	CASE iTagI OF
		1:
			IF i < DINT_TO_INT(UPPER_BOUND(stEmergencias, 1)) THEN
				RefEmer1 REF= stEmergencias[i].En.xEmergenciaOK;
			ELSE
				RefEmer1 REF= Verdadeiro;
			END_IF
		2:
			IF i < DINT_TO_INT(UPPER_BOUND(stEmergencias, 1)) THEN
				RefEmer2 REF= stEmergencias[i].En.xEmergenciaOK;
			ELSE
				RefEmer2 REF= Verdadeiro;
			END_IF		
		3:
			IF i < DINT_TO_INT(UPPER_BOUND(stEmergencias, 1)) THEN
				RefEmer3 REF= stEmergencias[i].En.xEmergenciaOK;
			ELSE
				RefEmer3 REF= Verdadeiro;
			END_IF
		4:
			IF i < DINT_TO_INT(UPPER_BOUND(stEmergencias, 1)) THEN
				RefEmer4 REF= stEmergencias[i].En.xEmergenciaOK;
			ELSE
				RefEmer4 REF= Verdadeiro;
			END_IF
		
	END_CASE
		
END_FOR

GeraEmergencias := TRUE;
END_METHOD

METHOD PRIVATE GeraNomeInterlock : BOOL
VAR_INPUT
	index : INT;
END_VAR
VAR
	sAux : ARRAY[1..20] OF STRING(255);
	i : INT;
END_VAR


IF stMotor[index].BancoDeDados.IT1A <> '' THEN
	
	IF stMotor[index].BancoDeDados.InvIT1A <> 0 THEN
		IF __ISVALIDREF(RefIT1A) THEN		
			IF (RefIT1A) THEN
				sAux[1] := 'NF(';
			ELSE
				sAux[1] := '*NF*(';
			END_IF
		END_IF
	ELSE
		IF __ISVALIDREF(RefIT1A) THEN	
			IF (RefIT1A) THEN
				sAux[1] := '*NA*(';
			ELSE
				sAux[1] := 'NA(';
			END_IF
		END_IF
	END_IF
	
	IF __ISVALIDREF(RefIT1A) THEN	
		IF (RefIT1A) THEN
			sAux[2] := CONCAT(CONCAT('*',(stMotor[index].BancoDeDados.IT1A)),'*');
		ELSE
			sAux[2] := (stMotor[index].BancoDeDados.IT1A);
		END_IF
	END_IF
	
	sAux[3] := 	')';

	IF stMotor[index].BancoDeDados.IT1B <> '' THEN
		IF stMotor[index].BancoDeDados.OPIT1 <> 0 THEN
			sAux[4] := ' E ';
		ELSE
			sAux[4] := 	' OU ';
		END_IF

		IF stMotor[index].BancoDeDados.InvIT1B <> 0 THEN
			IF __ISVALIDREF(RefIT1B) THEN
				IF (RefIT1B) THEN
					sAux[5] := 'NF(';
				ELSE
					sAux[5] := '*NF*(';
				END_IF
			END_IF
		ELSE
			IF __ISVALIDREF(RefIT1B) THEN
				IF (RefIT1B) THEN
					sAux[5] := '*NA*(';
				ELSE
					sAux[5] := 'NA(';
				END_IF
			END_IF
		END_IF
		
		IF __ISVALIDREF(RefIT1B) THEN
			IF (RefIT1B) THEN
				sAux[6] := CONCAT(CONCAT('*',(stMotor[index].BancoDeDados.IT1B)),'*');
			ELSE
				sAux[6] := (stMotor[index].BancoDeDados.IT1B);
			END_IF
		END_IF
		sAux[7] := 	') ';
	END_IF
ELSE
	stMotor[index].En.sInterLock_1 := '';
END_IF

stMotor[index].En.sInterLock_1 := F_ConcatArray(sAux);

FOR i := 1 TO 20 DO
	sAux[i] := '';
END_FOR


IF stMotor[index].BancoDeDados.IT2A <> '' THEN
	
	IF stMotor[index].BancoDeDados.InvIT2A <> 0 THEN
		IF __ISVALIDREF(RefIT2A) THEN		
			IF (RefIT2A) THEN
				sAux[1] := 'NF(';
			ELSE
				sAux[1] := '*NF*(';
			END_IF
		END_IF
	ELSE
		IF __ISVALIDREF(RefIT2A) THEN	
			IF (RefIT2A) THEN
				sAux[1] := '*NA*(';
			ELSE
				sAux[1] := 'NA(';
			END_IF
		END_IF
	END_IF
	
	IF __ISVALIDREF(RefIT2A) THEN	
		IF (RefIT2A) THEN
			sAux[2] := CONCAT(CONCAT('*',(stMotor[index].BancoDeDados.IT2A)),'*');
		ELSE
			sAux[2] := (stMotor[index].BancoDeDados.IT2A);
		END_IF
	END_IF
	
	sAux[3] := 	')';

	IF stMotor[index].BancoDeDados.IT2B <> '' THEN
		IF stMotor[index].BancoDeDados.OPIT2 <> 0 THEN
			sAux[4] := ' E ';
		ELSE
			sAux[4] := 	' OU ';
		END_IF

		IF stMotor[index].BancoDeDados.InvIT2B <> 0 THEN
			IF __ISVALIDREF(RefIT2B) THEN
				IF (RefIT2B) THEN
					sAux[5] := 'NF(';
				ELSE
					sAux[5] := '*NF*(';
				END_IF
			END_IF
		ELSE
			IF __ISVALIDREF(RefIT2B) THEN
				IF (RefIT2B) THEN
					sAux[5] := '*NA*(';
				ELSE
					sAux[5] := 'NA(';
				END_IF
			END_IF
		END_IF
		
		IF __ISVALIDREF(RefIT2B) THEN
			IF (RefIT2B) THEN
				sAux[6] := CONCAT(CONCAT('*',(stMotor[index].BancoDeDados.IT2B)),'*');
			ELSE
				sAux[6] := (stMotor[index].BancoDeDados.IT2B);
			END_IF
		END_IF
		sAux[7] := 	') ';
	END_IF
ELSE
	stMotor[index].En.sInterLock_2 := '';
END_IF

stMotor[index].En.sInterLock_2 := F_ConcatArray(sAux);

FOR i := 1 TO 20 DO
	sAux[i] := '';
END_FOR


IF stMotor[index].BancoDeDados.IT3A <> '' THEN
	
	IF stMotor[index].BancoDeDados.InvIT3A <> 0 THEN
		IF __ISVALIDREF(RefIT3A) THEN		
			IF (RefIT3A) THEN
				sAux[1] := 'NF(';
			ELSE
				sAux[1] := '*NF*(';
			END_IF
		END_IF
	ELSE
		IF __ISVALIDREF(RefIT3A) THEN	
			IF (RefIT3A) THEN
				sAux[1] := '*NA*(';
			ELSE
				sAux[1] := 'NA(';
			END_IF
		END_IF
	END_IF
	
	IF __ISVALIDREF(RefIT3A) THEN	
		IF (RefIT3A) THEN
			sAux[2] := CONCAT(CONCAT('*',(stMotor[index].BancoDeDados.IT3A)),'*');
		ELSE
			sAux[2] := (stMotor[index].BancoDeDados.IT3A);
		END_IF
	END_IF
	
	sAux[3] := 	')';

	IF stMotor[index].BancoDeDados.IT3B <> '' THEN
		IF stMotor[index].BancoDeDados.OPIT3 <> 0 THEN
			sAux[4] := ' E ';
		ELSE
			sAux[4] := 	' OU ';
		END_IF

		IF stMotor[index].BancoDeDados.InvIT3B <> 0 THEN
			IF __ISVALIDREF(RefIT3B) THEN
				IF (RefIT3B) THEN
					sAux[5] := 'NF(';
				ELSE
					sAux[5] := '*NF*(';
				END_IF
			END_IF
		ELSE
			IF __ISVALIDREF(RefIT3B) THEN
				IF (RefIT3B) THEN
					sAux[5] := '*NA*(';
				ELSE
					sAux[5] := 'NA(';
				END_IF
			END_IF
		END_IF
		
		IF __ISVALIDREF(RefIT3B) THEN
			IF (RefIT3B) THEN
				sAux[6] := CONCAT(CONCAT('*',(stMotor[index].BancoDeDados.IT3B)),'*');
			ELSE
				sAux[6] := (stMotor[index].BancoDeDados.IT3B);
			END_IF
		END_IF
		sAux[7] := 	') ';
	END_IF
ELSE
	stMotor[index].En.sInterLock_3 := '';
END_IF

stMotor[index].En.sInterLock_3 := F_ConcatArray(sAux);

FOR i := 1 TO 20 DO
	sAux[i] := '';
END_FOR


IF stMotor[index].BancoDeDados.IT4A <> '' THEN
	
	IF stMotor[index].BancoDeDados.InvIT4A <> 0 THEN
		IF __ISVALIDREF(RefIT4A) THEN		
			IF (RefIT4A) THEN
				sAux[1] := 'NF(';
			ELSE
				sAux[1] := '*NF*(';
			END_IF
		END_IF
	ELSE
		IF __ISVALIDREF(RefIT4A) THEN	
			IF (RefIT4A) THEN
				sAux[1] := '*NA*(';
			ELSE
				sAux[1] := 'NA(';
			END_IF
		END_IF
	END_IF
	
	IF __ISVALIDREF(RefIT4A) THEN	
		IF (RefIT4A) THEN
			sAux[2] := CONCAT(CONCAT('*',(stMotor[index].BancoDeDados.IT4A)),'*');
		ELSE
			sAux[2] := (stMotor[index].BancoDeDados.IT4A);
		END_IF
	END_IF
	
	sAux[3] := 	')';

	IF stMotor[index].BancoDeDados.IT4B <> '' THEN
		IF stMotor[index].BancoDeDados.OPIT4 <> 0 THEN
			sAux[4] := ' E ';
		ELSE
			sAux[4] := 	' OU ';
		END_IF

		IF stMotor[index].BancoDeDados.InvIT4B <> 0 THEN
			IF __ISVALIDREF(RefIT4B) THEN
				IF (RefIT4B) THEN
					sAux[5] := 'NF(';
				ELSE
					sAux[5] := '*NF*(';
				END_IF
			END_IF
		ELSE
			IF __ISVALIDREF(RefIT4B) THEN
				IF (RefIT4B) THEN
					sAux[5] := '*NA*(';
				ELSE
					sAux[5] := 'NA(';
				END_IF
			END_IF
		END_IF
		
		IF __ISVALIDREF(RefIT4B) THEN
			IF (RefIT4B) THEN
				sAux[6] := CONCAT(CONCAT('*',(stMotor[index].BancoDeDados.IT4B)),'*');
			ELSE
				sAux[6] := (stMotor[index].BancoDeDados.IT4B);
			END_IF
		END_IF
		sAux[7] := 	') ';
	END_IF
ELSE
	stMotor[index].En.sInterLock_4 := '';
END_IF

stMotor[index].En.sInterLock_4 := F_ConcatArray(sAux);

FOR i := 1 TO 20 DO
	sAux[i] := '';
END_FOR







GeraNomeInterlock := true;
END_METHOD

METHOD PRIVATE LinkaOsNaoInterlock : BOOL
VAR_INPUT
END_VAR
//Se inverte
IF EstruturaBanco[0].InvIT1A = 1 THEN
	RefInvIT1A REF= Verdadeiro;
ELSE
	RefInvIT1A REF= FALSO;
END_IF

//Operação feita
IF EstruturaBanco[0].OPIT1 = 1 THEN
	RefOPIT1 REF= Verdadeiro;
ELSE
	RefOPIT1 REF= FALSO;
END_IF

//Se inverte o 1B
IF EstruturaBanco[0].InvIT1B = 1 THEN
	RefInvIT1B REF= Verdadeiro;
ELSE
	RefInvIT1B REF= FALSO;
END_IF

//Se inverte
IF EstruturaBanco[0].InvIT2A = 1 THEN
	RefInvIT2A REF= Verdadeiro;
ELSE
	RefInvIT2A REF= FALSO;
END_IF

//Operação feita
IF EstruturaBanco[0].OPIT2 = 1 THEN
	RefOPIT2 REF= Verdadeiro;
ELSE
	RefOPIT2 REF= FALSO;
END_IF

//Se inverte o 2B
IF EstruturaBanco[0].InvIT2B = 1 THEN
	RefInvIT2B REF= Verdadeiro;
ELSE
	RefInvIT2B REF= FALSO;
END_IF

//Se inverte
IF EstruturaBanco[0].InvIT3A = 1 THEN
	RefInvIT3A REF= Verdadeiro;
ELSE
	RefInvIT3A REF= FALSO;
END_IF

//Operação feita
IF EstruturaBanco[0].OPIT3 = 1 THEN
	RefOPIT3 REF= Verdadeiro;
ELSE
	RefOPIT3 REF= FALSO;
END_IF

//Se inverte o 3B
IF EstruturaBanco[0].InvIT3B = 1 THEN
	RefInvIT3B REF= Verdadeiro;
ELSE
	RefInvIT3B REF= FALSO;
END_IF

//Se inverte
IF EstruturaBanco[0].InvIT4A = 1 THEN
	RefInvIT4A REF= Verdadeiro;
ELSE
	RefInvIT4A REF= FALSO;
END_IF

//Operação feita
IF EstruturaBanco[0].OPIT4 = 1 THEN
	RefOPIT4 REF= Verdadeiro;
ELSE
	RefOPIT4 REF= FALSO;
END_IF

//Se inverte o 4B
IF EstruturaBanco[0].InvIT4B = 1 THEN
	RefInvIT4B REF= Verdadeiro;
ELSE
	RefInvIT4B REF= FALSO;
END_IF
END_METHOD

METHOD PRIVATE MudouNoMotor : BOOL
VAR_INPUT
	Atual		: Teknike_Partidas.ST_ConfigMotorDB;
	Anterior	: Teknike_Partidas.ST_ConfigMotorDB;
END_VAR
VAR
	xMudouNome : BOOL;
	iTamanhoComecaFuncao : INT;
END_VAR

xMudouNome := (CONCAT(CONCAT(stMotor[iIndexMotor].BancoDeDados.Tag, ' - '), stMotor[iIndexMotor].BancoDeDados.Funcao))
				<> stMotor[iIndexMotor].Config.sNome_Funcao;

IF xMudouNome AND NOT (Anterior.Tag <> Atual.Tag OR ((Anterior.Funcao <> Atual.Funcao) AND Atual.Funcao <> '')) THEN
	IF (Anterior.Funcao <> Atual.Funcao) AND (Atual.Funcao = '' OR stMotor[iIndexMotor].Config.sNome_Funcao = '') THEN
		stMotor[iIndexMotor].Config.sNome_Funcao := concat(stMotor[iIndexMotor].BancoDeDados.Tag,stMotor[iIndexMotor].BancoDeDados.Funcao);
	END_IF
	iTamanhoComecaFuncao								:= LEN(stMotor[iIndexMotor].Config.sNome_Funcao) - (LEN(Atual.Tag) + 3);
	stMotor[iIndexMotor].BancoDeDados.Funcao	:= RIGHT(STR := stMotor[iIndexMotor].Config.sNome_Funcao, SIZE := iTamanhoComecaFuncao);
END_IF

MudouNoMotor := 	Anterior.InvIT1A <> Atual.InvIT1A
					OR Anterior.IT1A <> Atual.IT1A
					OR Anterior.OPIT1 <> Atual.OPIT1
					OR Anterior.InvIT1B <> Atual.InvIT1B
					OR Anterior.IT1B <> Atual.IT1B
					OR Anterior.InvIT2A <> Atual.InvIT2A
					OR Anterior.IT2A <> Atual.IT2A
					OR Anterior.OPIT2 <> Atual.OPIT2
					OR Anterior.InvIT2B <> Atual.InvIT2B
					OR Anterior.IT2B <> Atual.IT2B
					OR Anterior.InvIT3A <> Atual.InvIT3A
					OR Anterior.IT3A <> Atual.IT3A
					OR Anterior.OPIT3 <> Atual.OPIT3
					OR Anterior.InvIT3B <> Atual.InvIT3B
					OR Anterior.IT3B <> Atual.IT3B
					OR Anterior.InvIT4A <> Atual.InvIT4A
					OR Anterior.IT4A <> Atual.IT4A
					OR Anterior.OPIT4 <> Atual.OPiT4
					OR Anterior.InvIT4B <> Atual.InvIT4B
					OR Anterior.IT4B <> Atual.IT4B
					OR Anterior.Emerg1 <> Atual.Emerg1
					OR Anterior.Emerg2 <> Atual.Emerg2
					OR Anterior.Emerg3 <> Atual.Emerg3
					OR Anterior.Emerg4 <> Atual.Emerg4
					OR xMudouNome;
END_METHOD

ACTION TrocaEstadoLeitura:

//EstadoAtual := ExecutaInterlocks;

CASE EstadoAtual OF

	enum_MaquinaConfigPartidaDB.Esperando:
		xOcupado := FALSE;
		rtAtualiza(CLK := xLe, Q =>);

		//controla pra nao ficar muitos acessando o banco 
		//IF rtAtualiza.q THEN
			IF iMaxAtualizando > iAtualizandoAtual AND xLe THEN
				EstadoAtual	:= enum_MaquinaConfigPartidaDB.LendoEleMesmo;
				xOcupado	:= TRUE;
			//ELSE
			//	xLe := FALSE;
			END_IF	
		//END_IF

		EstruturaAnterior := stMotor[iIndexMotor].BancoDeDados;

	enum_MaquinaConfigPartidaDB.AbreConexao:
		//xOcupado := TRUE;
		
		xTemQueAtualizarSQL := FALSE;//joga pra falso pq so aqui é que realmente ele ta atualizando o SQL
		
		IF fbSqlDatabase.Connect(INT_TO_UDINT(iNumeroDataBase)) THEN
			IF fbSqlDatabase.bError THEN
				{error <'Não conseguiu conectar para ler o banco no bloco FB_ConfigPartidaNoBanco 1'>}
				IF fbSqlDatabase.ipTcResult.nEventId = 1828 THEN
					// se der isso ele nao fica tentando e gerando uma caralhada de erro pq nao tem a lisença
					EstadoAtual := enum_MaquinaConfigPartidaDB.falha;
				ELSE
					EstadoAtual := enum_MaquinaConfigPartidaDB.AbreConexao;
				END_IF
			ELSE
				IF fbSqlDatabase.bConnected THEN
					EstadoAtual := enum_MaquinaConfigPartidaDB.CriaComando;
				END_IF
			END_IF
		END_IF

	enum_MaquinaConfigPartidaDB.CriaComando:
		//xOcupado := TRUE;

		IF fbSqlDatabase.CreateCmd(ADR(fbSqlCommand)) THEN
			IF fbSqlDatabase.bError THEN
				{error <'Não conseguiu criar o comando para ler o banco no bloco FB_ConfigPartidaNoBanco 2'>}
				EstadoAtual := enum_MaquinaConfigPartidaDB.CriaComando;
			ELSE
				EstadoAtual := enum_MaquinaConfigPartidaDB.Gravando;
			END_IF
		END_IF

	enum_MaquinaConfigPartidaDB.Gravando:
		//xOcupado := TRUE;

		IF sCmdUpdate <> '' THEN
			IF fbSQLCommand.Execute(pSQLCmd := ADR(sCmdUpdate), cbSQLCmd := SIZEOF(sCmdUpdate)) THEN
				EstadoAtual	:= enum_MaquinaConfigPartidaDB.FechaConexao;
				sCmdUpdate	:= '';
			END_IF
		END_IF

	enum_MaquinaConfigPartidaDB.FechaConexao:
		//xOcupado := TRUE;

		IF fbSqlDatabase.Disconnect() THEN
			IF fbSqlDatabase.bError THEN
				{error <'Não conseguiu desconectar depois de ler o banco no bloco FB_ConfigPartidaNoBanco 3'>}
				EstadoAtual := enum_MaquinaConfigPartidaDB.FechaConexao;
			ELSE
				xLe			:= TRUE;
				EstadoAtual	:= enum_MaquinaConfigPartidaDB.LendoEleMesmo;
			END_IF
		END_IF

	enum_MaquinaConfigPartidaDB.LendoEleMesmo:
		//xOcupado := TRUE;

		IF NOT xLe THEN
			EstadoAtual := enum_MaquinaConfigPartidaDB.LinkaOsNaoInterlock;
		END_IF

	enum_MaquinaConfigPartidaDB.LinkaOsNaoInterlock:
		//xOcupado			:= TRUE;

		IF __ISVALIDREF(RefInvIT4A) AND __ISVALIDREF(RefOPIT4) AND __ISVALIDREF(RefInvIT4B) THEN
			EstadoAtual	:= enum_MaquinaConfigPartidaDB.ProcuraTag1;
			iTag		:= 1;
		END_IF

	enum_MaquinaConfigPartidaDB.ProcuraTag1:
		//xOcupado			:= TRUE;

		IF __ISVALIDREF(RefIT1A) AND __ISVALIDREF(RefIT2A) AND __ISVALIDREF(RefIT3A) AND __ISVALIDREF(RefIT4A) THEN
			EstadoAtual	:= enum_MaquinaConfigPartidaDB.ProcuraTag2;
			iTag		:= 1;
		END_IF

	enum_MaquinaConfigPartidaDB.ProcuraTag2:
		//xOcupado			:= TRUE;

		IF __ISVALIDREF(RefIT1B) AND __ISVALIDREF(RefIT2B) AND __ISVALIDREF(RefIT3B) AND __ISVALIDREF(RefIT4B) THEN
			EstadoAtual := enum_MaquinaConfigPartidaDB.Gera_sInterlock;
		END_IF

	enum_MaquinaConfigPartidaDB.Gera_sInterlock:
		//xOcupado			:= TRUE;
		EstruturaAnterior	:= stMotor[iIndexMotor].BancoDeDados;
		
		stMotor[iIndexMotor].Config.sNome_Funcao := (CONCAT(CONCAT(stMotor[iIndexMotor].BancoDeDados.Tag,' - '),stMotor[iIndexMotor].BancoDeDados.Funcao));

		IF GeraNomeInterlock(iIndexMotor) THEN
			EstadoAtual := enum_MaquinaConfigPartidaDB.Gera_Emergencia;
		END_IF
		
	enum_MaquinaConfigPartidaDB.Gera_Emergencia:
		IF GeraEmergencias(iIndexMotor) THEN
			EstadoAtual := enum_MaquinaConfigPartidaDB.ExecutaInterlocks;
		END_IF

	enum_MaquinaConfigPartidaDB.ExecutaInterlocks:
		xOcupado := FALSE;
		
		GeraNomeInterlock(iIndexMotor);
		
		rtAtualiza(CLK := xLe, Q =>);

		//controla pra nao ficar muitos acessando o banco 
		IF iMaxAtualizando > iAtualizandoAtual AND xLe THEN
			EstadoAtual	:= enum_MaquinaConfigPartidaDB.LendoEleMesmo;
			xOcupado	:= TRUE;	
		END_IF

		IF xAtualizadoExternamente THEN
			xAtualizadoExternamente	:= FALSE;
			GeraNomeInterlock(iIndexMotor);
			stMotor[iIndexMotor].Config.sNome_Funcao := (CONCAT(CONCAT(stMotor[iIndexMotor].BancoDeDados.Tag,' - '),stMotor[iIndexMotor].BancoDeDados.Funcao));
			EstruturaAnterior		:= stMotor[iIndexMotor].BancoDeDados;
		END_IF
		
		IF MudouNoMotor(stMotor[iIndexMotor].BancoDeDados, EstruturaAnterior) THEN
			xTemQueAtualizarSQL := TRUE;
		END_IF

		IF xTemQueAtualizarSQL AND iMaxAtualizando > iAtualizandoAtual THEN
			EstadoAtual	:= enum_MaquinaConfigPartidaDB.AbreConexao;
			xOcupado	:= TRUE;
		END_IF

		//EstruturaAnterior := stMotor[iIndexMotor].BancoDeDados;

END_CASE
END_ACTION

METHOD PRIVATE ZeraReferencias : BOOL
VAR_INPUT
END_VAR


RefInvIT1A	REF= 0;
IF stMotor[iIndexMotor].BancoDeDados.IT1A <> EstruturaAnterior.IT1A THEN
	RefIT1A	REF= 0;
END_IF
RefOPIT1	REF= 0;
RefInvIT1B	REF= 0;
IF stMotor[iIndexMotor].BancoDeDados.IT1B <> EstruturaAnterior.IT1B THEN
	RefIT1B	REF= 0;
END_IF

RefInvIT2A	REF= 0;
IF stMotor[iIndexMotor].BancoDeDados.IT2A <> EstruturaAnterior.IT2A THEN
	RefIT2A	REF= 0;
END_IF
RefOPIT2	REF= 0;
RefInvIT2B	REF= 0;
IF stMotor[iIndexMotor].BancoDeDados.IT2B <> EstruturaAnterior.IT2B THEN
	RefIT2B	REF= 0;
END_IF

RefInvIT3A	REF= 0;
IF stMotor[iIndexMotor].BancoDeDados.IT3A <> EstruturaAnterior.IT3A THEN
	RefIT3A	REF= 0;
END_IF
RefOPIT3	REF= 0;
RefInvIT3B	REF= 0;
IF stMotor[iIndexMotor].BancoDeDados.IT3B <> EstruturaAnterior.IT3B THEN
	RefIT3B	REF= 0;
END_IF

RefInvIT4A	REF= 0;
IF stMotor[iIndexMotor].BancoDeDados.IT4A <> EstruturaAnterior.IT4A THEN
	RefIT4A	REF= 0;
END_IF
RefOPIT4	REF= 0;
RefInvIT4B	REF= 0;
IF stMotor[iIndexMotor].BancoDeDados.IT4B <> EstruturaAnterior.IT4B THEN
	RefIT4B	REF= 0;
END_IF


RefEmer1	REF= 0;
RefEmer2	REF= 0;
RefEmer3	REF= 0;
RefEmer4	REF= 0;
END_METHOD

END_FUNCTION_BLOCK

// FBs/Intralogistica/Top10SKU/FB_HistogramaSKUsMaisLidas
//{attribute 'hide_all_locals'}
FUNCTION_BLOCK FB_HistogramaSKUsMaisLidas
VAR_INPUT
	sSKU			: STRING;
	xEscreve 		: BOOL;
	xCriaEvento		: BOOL := TRUE;
	xVeOsTop10		: BOOL;
	TempoGuardandoSKUemMinutos : UDINT := 60;
	xCriaTabela		: BOOL;
	iNumeroDataBase	: INT := 1;
	sNomeTabela		: STRING	:= 'TopSKU';
END_VAR
VAR_OUTPUT
	TopSKUs 			: ARRAY[1..10] OF DUT_Top10SKU;
	EstadoEscreve 		: Enum_HistorogramaSKUs := Enum_HistorogramaSKUs.Esperando;
	EstadoEvento 		: Enum_HistorogramaSKUs := Enum_HistorogramaSKUs.Esperando;
	EstadoTOP 			: Enum_HistorogramaSKUs := Enum_HistorogramaSKUs.Esperando;
END_VAR
VAR
	UltimotempoGuardado : UDINT;
	rtCria			: R_TRIG;
	xCria			: BOOL;
	fbPLCDBCreate	: FB_PLCDBCreateEvt(sNetID := '', tTimeout := T#30S);

	ColumnInfo : ARRAY[0..2] OF ST_ColumnInfo := [(sName := 'ID', eType := E_ColumnType.BigInt, nLength := 8, sProperty := 'IDENTITY(1,1)'),
												(sName := 'SKU', eType := E_ColumnType.Integer, nLength := 4),
												(
				sName := 'Timestamp',
					eType := E_ColumnType.DateTime,
					nLength := 4,
					sProperty := 'DEFAULT CURRENT_TIMESTAMP ON UPDATE CURRENT_TIMESTAMP')];



	ColumnNamesLe : ARRAY[0..2] OF STRING(50) := ['ID',
												'SKU',
												'Timestamp'];
	iTamanhoHistorico : DINT;

	i : INT;
	
	fbSqlCommandEscreve		: FB_SQLCommandEvt(sNetID := '', tTimeout := T#30S);
	fbSQLDatabaseEscreve	: FB_SQLDatabaseEvt(sNetID := '', tTimeout := T#30S);
	sCmdEscreve				: STRING(1000);
	xAbertoEscreve 			: BOOL;
	rtEscreve 				: R_TRIG;
	sAuxEscreve				: ARRAY[0..10] OF STRING(255);
	
	fbSqlCommandEvento		: FB_SQLCommandEvt(sNetID := '', tTimeout := T#30S);
	fbSQLDatabaseEvento		: FB_SQLDatabaseEvt(sNetID := '', tTimeout := T#30S);
	sCmdEvento				: STRING(1000);
	xAbertoEvento 			: BOOL;
	rtEvento 				: R_TRIG;
	sAuxEvento				: ARRAY[0..10] OF STRING(255);
	
	
	fbSqlCommandtop			: FB_PLCDBCmdEvt(sNetID := '', tTimeout := T#30S);
	fbSQLDatabaseTOP		: FB_SQLDatabaseEvt(sNetID := '', tTimeout := T#30S);
	sCmdTOP					: STRING(1000);
	xAbertoTOP 				: BOOL;
	rtTOP 					: R_TRIG;
	sAuxTop					: ARRAY[0..10] OF STRING(255);
	stParaTop				: ST_ExpParameter;
	sPara					: STRING(80);
	nRecords				: UDINT;
	LeituraAux				: ARRAY[1..10] OF DUT_Top10SKU;
	
	sMensagemErro1 		: STRING;
	rtComecaEscrever : R_TRIG;
	

END_VAR


IF xLicensaValida651641iih THEN
	
	rtEscreve(CLK:= xEscreve, Q=> );
	rtEvento(CLK:= xCriaEvento OR TempoGuardandoSKUemMinutos <> UltimotempoGuardado, Q=> );
	rtTop(CLK:= xVeOsTop10, Q=> );
	
	UltimotempoGuardado := TempoGuardandoSKUemMinutos;
	
	GeraTabela();
	
	Tabela();
	
	Evento();
	
	Top10();

END_IF

ACTION Evento:

CASE EstadoEvento OF
	 Enum_HistorogramaSKUs.Esperando: //Esperando
		IF rtEvento.q THEN
			IF xAbertoEvento THEN
				EstadoEvento := Enum_HistorogramaSKUs.CriaComando;
			ELSE
				EstadoEvento := Enum_HistorogramaSKUs.AbreConexao;
			END_IF
		END_IF

	Enum_HistorogramaSKUs.AbreConexao: //abre conexao
		IF fbSQLDatabaseEvento.Connect(int_to_udint(iNumeroDataBase)) THEN
			IF fbSQLDatabaseEvento.bError THEN
				IF fbSQLDatabaseEvento.ipTcResult.nEventId = 1828 THEN
					// se der isso ele nao fica tentando e gerando uma caralhada de erro pq nao tem a lisensa
					EstadoEvento := Enum_HistorogramaSKUs.erro;
				ELSE
					EstadoEvento := Enum_HistorogramaSKUs.AbreConexao;
				END_IF
			ELSE
				IF fbSQLDatabaseEvento.bConnected THEN
					EstadoEvento := Enum_HistorogramaSKUs.CriaComando;
					xAbertoEvento := TRUE;
				ELSE
					EstadoEvento := Enum_HistorogramaSKUs.FechaConexao;
					xAbertoEvento := FALSE;
				END_IF
			END_IF
		END_IF
	
	Enum_HistorogramaSKUs.CriaComando:
		IF fbSQLDatabaseEvento.CreateCmd(ADR(fbSqlCommandEvento)) THEN
			IF fbSQLDatabaseEvento.bError THEN
				EstadoEvento := Enum_HistorogramaSKUs.CriaComando;
			ELSE
				EstadoEvento := Enum_HistorogramaSKUs.DeletaEvento;
			END_IF
		END_IF
	
		
	Enum_HistorogramaSKUs.DeletaEvento:
	
		F_LimpaArrayString(sAuxEvento);
	
		sAuxEvento[0] := 'drop event Exclui';
		sAuxEvento[1] := sNomeTabela;
		sAuxEvento[2] := ';';

		sCmdEvento := F_ConcatArray(sAuxEvento);	


		// call functionblock	
		IF fbSqlCommandEvento.Execute(pSQLCmd := ADR(sCmdEvento), cbSQLCmd := SIZEOF(sCmdEvento))THEN
			IF fbSqlCommandEvento.bError THEN
				IF fbSqlCommandEvento.ipTcResult.nEventId = 61 THEN
				// se der isso ele nao fica tentando e gerando uma caralhada de erro pq nao tem a tabela
					EstadoEvento := Enum_HistorogramaSKUs.Esperando;
					xCriaTabela := TRUE;
				ELSE
					EstadoEvento := Enum_HistorogramaSKUs.DeletaEvento;
				END_IF
				sMensagemErro1 := 'Nao conseguiu a tag';
			ELSE
				sMensagemErro1	:= 'Conseguiu a tag';
			END_IF
			EstadoEvento := Enum_HistorogramaSKUs.CriaEvento;
		END_IF
		
	Enum_HistorogramaSKUs.CriaEvento:
	
		F_LimpaArrayString(sAuxEvento);
	
		sAuxEvento[0] := 'CREATE EVENT IF NOT EXISTS Exclui';
		sAuxEvento[1] := sNomeTabela;
		sAuxEvento[2] := ' ON SCHEDULE every 1 minute DO delete from topsku where Timestamp < (NOW() - interval ';
		sAuxEvento[3] := UDINT_TO_STRING(TempoGuardandoSKUemMinutos);
		sAuxEvento[4] := ' minute);';

		 

		sCmdEvento := F_ConcatArray(sAuxEvento);	


		// call functionblock	
		IF fbSqlCommandEvento.Execute(pSQLCmd := ADR(sCmdEvento), cbSQLCmd := SIZEOF(sCmdEvento))THEN
			IF fbSqlCommandEvento.bError THEN
				IF fbSqlCommandEvento.ipTcResult.nEventId = 61 THEN
				// se der isso ele nao fica tentando e gerando uma caralhada de erro pq nao tem a tabela
					EstadoEvento := Enum_HistorogramaSKUs.Esperando;
					xCriaTabela := TRUE;
				ELSE
					EstadoEvento := Enum_HistorogramaSKUs.CriaEvento;
				END_IF
				sMensagemErro1 := 'Nao conseguiu a tag';
			ELSE
				sMensagemErro1	:= 'Conseguiu a tag';
			END_IF
			EstadoEvento := Enum_HistorogramaSKUs.FechaConexao;
			xCriaEvento := FALSE;
		END_IF
		

	Enum_HistorogramaSKUs.FechaConexao: // FechaConexao conexao
		IF fbSQLDatabaseEvento.Disconnect() THEN
			IF NOT fbSQLDatabaseEvento.bError THEN
				EstadoEvento := Enum_HistorogramaSKUs.Esperando;
				xAbertoEvento := FALSE;
			END_IF
		END_IF
END_CASE
END_ACTION

ACTION GeraTabela:

rtCria(CLK := xCriaTabela, Q =>);

IF rtCria.q THEN
	xCria := TRUE;
END_IF

IF xCria THEN
	IF fbPLCDBCreate.Table(
			hDBID := INT_TO_UDINT(iNumeroDataBase),
			sTableName := sNomeTabela,
			pTableCfg := ADR(ColumnInfo),
			cbTableCfg := SIZEOF(ColumnInfo))
	THEN
		xCria := FALSE;
		xCriaTabela := FALSE;
	END_IF

END_IF
END_ACTION

ACTION Tabela:

CASE EstadoEscreve OF
	Enum_HistorogramaSKUs.Esperando: //Esperando
		IF rtEscreve.q THEN
			IF xAbertoEscreve THEN
				EstadoEscreve := Enum_HistorogramaSKUs.CriaComando;
			ELSE
				EstadoEscreve := Enum_HistorogramaSKUs.AbreConexao;
			END_IF
		END_IF

	Enum_HistorogramaSKUs.AbreConexao: //abre conexao
		IF fbSQLDatabaseEscreve.Connect(int_to_udint(iNumeroDataBase)) THEN
			IF fbSQLDatabaseEscreve.bError THEN
				IF fbSQLDatabaseEscreve.ipTcResult.nEventId = 1828 THEN
					// se der isso ele nao fica tentando e gerando uma caralhada de erro pq nao tem a lisensa
					EstadoEscreve := Enum_HistorogramaSKUs.erro;
				ELSE
					EstadoEscreve := Enum_HistorogramaSKUs.AbreConexao;
				END_IF
			ELSE
				IF fbSQLDatabaseEscreve.bConnected THEN
					EstadoEscreve := Enum_HistorogramaSKUs.CriaComando;
					xAbertoEscreve := TRUE;
				ELSE
					EstadoEscreve := Enum_HistorogramaSKUs.FechaConexao;
					xAbertoEscreve := FALSE;
				END_IF
			END_IF
		END_IF
	
	Enum_HistorogramaSKUs.CriaComando:
		IF fbSQLDatabaseEscreve.CreateCmd(ADR(fbSqlCommandEscreve)) THEN
			IF fbSQLDatabaseEscreve.bError THEN
				EstadoEscreve := Enum_HistorogramaSKUs.CriaComando;
			ELSE
				EstadoEscreve := Enum_HistorogramaSKUs.Grava;
			END_IF
		END_IF
	

	Enum_HistorogramaSKUs.Grava: // le o role
	
		F_LimpaArrayString(sAuxEscreve);
	
		sAuxEscreve[0] := 'INSERT INTO ';
		sAuxEscreve[1] := sNomeTabela;
		sAuxEscreve[2] := '(sku) Value ($'';
		sAuxEscreve[3] := sSKU;
		sAuxEscreve[4] := '$');';

		sCmdEscreve := F_ConcatArray(sAuxEscreve);	



		IF fbSqlCommandEscreve.Execute(pSQLCmd := ADR(sCmdEscreve), cbSQLCmd := SIZEOF(sCmdEscreve)) THEN
			IF fbSqlCommandEscreve.bError THEN
				IF fbSqlCommandEscreve.ipTcResult.nEventId = 61 THEN
				// se der isso ele nao fica tentando e gerando uma caralhada de erro pq nao tem a tabela
					EstadoEscreve := Enum_HistorogramaSKUs.Esperando;
					xCriaTabela := TRUE;
				ELSE
					EstadoEscreve := Enum_HistorogramaSKUs.AbreConexao;
				END_IF
				sMensagemErro1 := 'Nao conseguiu a tag';
			ELSE
				sMensagemErro1	:= 'Conseguiu a tag';
			END_IF
			EstadoEscreve := Enum_HistorogramaSKUs.FechaConexao;
			xEscreve := FALSE;
		END_IF
		
	
		

	Enum_HistorogramaSKUs.FechaConexao: // FechaConexao conexao
		IF fbSQLDatabaseEscreve.Disconnect() THEN
			IF NOT fbSQLDatabaseEscreve.bError THEN
				EstadoEscreve := Enum_HistorogramaSKUs.Esperando;
				xAbertoEscreve := FALSE;
			END_IF
		END_IF
END_CASE
END_ACTION

ACTION Top10:

CASE Estadotop OF
	Enum_HistorogramaSKUs.Esperando: //Esperando
		IF rtTop.q THEN
			IF xAbertoTop THEN
				Estadotop := Enum_HistorogramaSKUs.CriaComando;
			ELSE
				Estadotop := Enum_HistorogramaSKUs.AbreConexao;
			END_IF
		END_IF

	Enum_HistorogramaSKUs.AbreConexao: //abre conexao
		IF fbSQLDatabasetop.Connect(int_to_udint(iNumeroDataBase)) THEN
			IF fbSQLDatabasetop.bError THEN
				IF fbSQLDatabasetop.ipTcResult.nEventId = 1828 THEN
					// se der isso ele nao fica tentando e gerando uma caralhada de erro pq nao tem a lisensa
					Estadotop := Enum_HistorogramaSKUs.erro;
				ELSE
					Estadotop := Enum_HistorogramaSKUs.AbreConexao;
				END_IF
			ELSE
				IF fbSQLDatabasetop.bConnected THEN
					Estadotop := Enum_HistorogramaSKUs.Vetop10;
					xAbertotop := TRUE;
				ELSE
					Estadotop := Enum_HistorogramaSKUs.FechaConexao;
					xAbertotop := FALSE;
				END_IF
			END_IF
		END_IF
	
		
	Enum_HistorogramaSKUs.Vetop10:
	
		F_LimpaArrayString(sAuxtop);
	
		sAuxtop[0] := 'SELECT SKU, count(*) FROM ';
		sAuxtop[1] := sNomeTabela;
		sAuxtop[2] := ' GROUP BY SKU ORDER BY count(*) DESC LIMIT 10;';
		 
		sCmdtop := F_ConcatArray(sAuxtop);	
		
		
		stParaTop.eParaType	:= E_ExpParameterType.STRING_;
		stParaTop.nParaSize	:= SIZEOF(sPara);
		stParaTop.sParaName	:= 'Inutil';


		// call functionblock	
		IF fbSqlCommandtop.ExecuteDataReturn(
										hDBID := INT_TO_UDINT(iNumeroDataBase),
										pExpression := ADR(sCmdtop),
										cbExpression := SIZEOF(sCmdtop),
										pData := ADR(sPara),
										cbData := SIZEOF(sPara),
										pParameter := ADR(stParaTop),
										cbParameter := SIZEOF(stParaTop),
										nStartIndex := 0,
										nRecordCount := 10,
										pReturnData := ADR(TopSKUs),
										cbReturnData := SIZEOF(TopSKUs),
										pRecords := ADR(nRecords))
													THEN
			IF fbSqlCommandtop.bError THEN
				IF fbSqlCommandtop.ipTcResult.nEventId = 61 THEN
				// se der isso ele nao fica tentando e gerando uma caralhada de erro pq nao tem a tabela
					Estadotop := Enum_HistorogramaSKUs.Esperando;
					xCriaTabela := TRUE;
				ELSE
					Estadotop := Enum_HistorogramaSKUs.FechaConexao;
				END_IF
				sMensagemErro1 := 'Nao conseguiu a tag';
			ELSE
				sMensagemErro1	:= 'Conseguiu a tag';
			END_IF
			Estadotop := Enum_HistorogramaSKUs.FechaConexao;
			xVeOsTop10 := FALSE;
		END_IF
		

	Enum_HistorogramaSKUs.FechaConexao: // FechaConexao conexao
		IF fbSQLDatabasetop.Disconnect() THEN
			IF NOT fbSQLDatabasetop.bError THEN
				Estadotop := Enum_HistorogramaSKUs.Esperando;
				xAbertotop := FALSE;
			END_IF
		END_IF
END_CASE
END_ACTION

END_FUNCTION_BLOCK

// FBs/MedicaoEnergia/FB_CentroDeCustos2
FUNCTION_BLOCK FB_CentroDeCustos2
VAR_IN_OUT
	Minutos				: ARRAY[*] OF stMinuto;
	Media15Min			: ARRAY[*] OF stMedia15min;
	MediaDia			: ARRAY[*] OF stMediaDia;
	MediaMes			: ARRAY[*] OF stMediaMes;
	PosicaoAtualdos15	: ARRAY[*,*] OF INT;
END_VAR
VAR_INPUT
	xCriaTabelas			: BOOL;				// tenta criar a tabela
	iNumeroDataBase			: INT	:= 1;		// id do database
	iMedidor				: INT;
	sMedidor				: STRING(1000);
	Timestamp				: DT;
	xAtualiza				: BOOL;
	x15minSelecionado		: BOOL;
	xDiaSelecionado			: BOOL;
	xMesSelecionado			: BOOL;
	xAnoSelecionado			: BOOL;
END_VAR
VAR_OUTPUT
	xOcupado 				: BOOL;
	xTodasTabelasCriadas	: BOOL;
	xTerminouLeitura		: BOOL := FALSE;
	sMedidoresSelecionados	: STRING(1000);
END_VAR
VAR
	//Le Valores Centros de Custo
	xAtualizaInterno			: BOOL;
	sCmdEscreve1				: STRING(2000);
	sCmdEscreve2				: STRING(2000);
	sCmdEscreve3				: STRING(2000);
	sCmdEscreve4				: STRING(2000);
	sMensagemErro				: STRING;
	nRecords					: UDINT;
	TagAProcurar				: REAL;
	arString					: ARRAY[0..12] OF STRING(1000);
	diCima						: DINT;
	diBaixo						: DINT;
	i							: INT;
	j							: INT;
	posicao						: INT := 1;
	iEstadoLeitura				: INT := 1;
	minute						: TIMESTRUCT;
	times						: TIMESTRUCT;
	TagAProcurar2				: REAL;
	fbSQLDatabase2				: FB_SQLDatabaseEvt(sNetID := '', tTimeout := T#30S);
	fbPLCDBCmd1					: FB_PLCDBCmdEvt(sNetID := '', tTimeout := T#30S);
	fbPLCDBCmd2					: FB_PLCDBCmdEvt(sNetID := '', tTimeout := T#30S);
	fbPLCDBCmd3					: FB_PLCDBCmdEvt(sNetID := '', tTimeout := T#30S);
	fbPLCDBCmd4					: FB_PLCDBCmdEvt(sNetID := '', tTimeout := T#30S);
	stPara2						: ST_ExpParameter;
	MinutosAtuais				: ARRAY[1..15] OF INT;
	EstruturaBancoMinuto		: ARRAY[1..900] OF stMinuto;
	EstruturaBancoMedia15min	: ARRAY[1..5760] OF stMedia15min;
	EstruturaBancoMediaDia		: ARRAY[1..1860] OF stMediaDia;
	EstruturaBancoMediaMes		: ARRAY[1..720] OF stMediaMes;
	OrganizaEstrutura			: ARRAY[0..132] OF stOrganizaDados;
	rtLeitura1					: R_TRIG;
	rtLeitura2					: R_TRIG;
	rtLeitura3					: R_TRIG;
	rtLeitura4					: R_TRIG;
	rtLeitura5					: R_TRIG;
END_VAR

rtLeitura1(CLK:= xAtualiza, Q=> );
rtLeitura2(CLK:= x15minSelecionado, Q=> );
rtLeitura3(CLK:= xDiaSelecionado, Q=> );
rtLeitura4(CLK:= xMesSelecionado, Q=> );
rtLeitura5(CLK:= xAnoSelecionado, Q=> );

IF rtLeitura1.Q OR rtLeitura2.Q OR rtLeitura3.Q OR rtLeitura4.Q OR rtLeitura5.Q THEN
	xAtualizaInterno 	:= TRUE;
	xTerminouLeitura	:= FALSE;
END_IF

sMedidoresSelecionados := sMedidor;

LeValores();

ACTION LeValores:
CASE iEstadoLeitura OF
	1: //Esperando
		IF xAtualizaInterno THEN
			iEstadoLeitura := 2;
		END_IF

	2: //abre conexao
		IF fbSQLDatabase2.Connect(INT_TO_UDINT(iNumeroDataBase)) THEN
			IF fbSQLDatabase2.bError THEN
				IF fbSQLDatabase2.ipTcResult.ipSourceInfo.sName = 'ADSERR_DEVICE_LICENSENOTFOUND' THEN
					// se der isso ele nao fica tentando e gerando uma caralhada de erro pq nao tem a lisença
					iEstadoLeitura := 0;
				ELSE
					iEstadoLeitura := 2;
				END_IF
			ELSE
				IF fbSQLDatabase2.bConnected THEN
					iEstadoLeitura := 3;
				END_IF
			END_IF
		END_IF

	3: 
		IF x15minSelecionado THEN
			// Le os Minutos
			stPara2.eParaType	:= E_ExpParameterType.Float32;
			stPara2.nParaSize	:= SIZEOF(TagAProcurar);
			stPara2.sParaName	:= 'rDemanda1min';
			
			IF sMedidor = '' THEN
				sMedidor := '1';
			END_IF
			
			arString[0] := 'SELECT * FROM dbexcelsior.minutos WHERE medidor in (';
			arString[1] := sMedidor;
			arString[2] := ') AND timestamps BETWEEN ';
			arString[3] := CONCAT(CONCAT('("',RIGHT(STR:= DT_TO_STRING(Timestamp - T#3H), SIZE:= 19)),'"- INTERVAL 15 MINUTE)');
			arString[4] := ' AND ';
			arString[5] := CONCAT(CONCAT('("',RIGHT(STR:= DT_TO_STRING(Timestamp - T#3H), SIZE:= 19)), '");');
			
			CONCAT2(pSrcString1:= ADR(arString[0]), pSrcString2:= ADR(arString[1]), pDstString:= ADR(arString[6]), nDstSize:= SIZEOF(arString[6]));
			CONCAT2(pSrcString1:= ADR(arString[6]), pSrcString2:= ADR(arString[2]), pDstString:= ADR(arString[7]), nDstSize:= SIZEOF(arString[7]));
			CONCAT2(pSrcString1:= ADR(arString[7]), pSrcString2:= ADR(arString[3]), pDstString:= ADR(arString[8]), nDstSize:= SIZEOF(arString[8]));
			CONCAT2(pSrcString1:= ADR(arString[8]), pSrcString2:= ADR(arString[4]), pDstString:= ADR(arString[9]), nDstSize:= SIZEOF(arString[9]));
			CONCAT2(pSrcString1:= ADR(arString[9]), pSrcString2:= ADR(arString[5]), pDstString:= ADR(arString[10]), nDstSize:= SIZEOF(arString[10]));
			
			sCmdEscreve1 := arString[10];
			
			//Cria o array dos minutos e limpa o array atual
			FOR i := 1 TO 15 DO
				Minutos[i].Medidor := 0;
				Minutos[i].rDemanda1min := 0;
				Minutos[i].rConsumo1min := 0;
				Minutos[i].rFatorDePotencia1min := 0;
				Minutos[i].Timestamp := DT#1970-1-1-0:0:0;
			
				minute	:= DT_TO_SYSTEMTIME(Timestamp);
				MinutosAtuais[i] := WORD_TO_INT(minute.wMinute)-i+1;
				IF MinutosAtuais[i] < 0 THEN
					MinutosAtuais[i] := 60 + MinutosAtuais[i];
				END_IF
			END_FOR
			
			// call functionblock
			IF fbPLCDBCmd1.ExecuteDataReturn
				(
					hDBID := 1,
						pExpression := ADR(sCmdEscreve1),
						cbExpression := SIZEOF(sCmdEscreve1),
						pData := ADR(TagAProcurar2),
						cbData := SIZEOF(TagAProcurar2),
						pParameter := ADR(stPara2),
						cbParameter := SIZEOF(stPara2),
						nStartIndex := 0,
						nRecordCount := 900,
						pReturnData := ADR(EstruturaBancoMinuto),
						cbReturnData := SIZEOF(EstruturaBancoMinuto),
						pRecords := ADR(nRecords))
			THEN
				IF fbPLCDBCmd1.bError THEN
					sMensagemErro := 'Nao conseguiu a tag';
				ELSE
					sMensagemErro	:= 'Conseguiu a tag';

					//Organiza os dados
					FOR i := 1 TO 900 DO
  						FOR j:= 1 TO 15 DO
							//OrganizaEstrutura[EstruturaBancoMinuto[i].Medidor].minuto[j] := EstruturaBancoMinuto[i];
							minute	:= DT_TO_SYSTEMTIME(EstruturaBancoMinuto[i].Timestamp);
							IF (WORD_TO_INT(minute.wMinute) = MinutosAtuais[j] AND EstruturaBancoMinuto[i].Timestamp <> DT#1970-1-1-0:0:0) THEN
								Minutos[j].Medidor				:= Minutos[i].Medidor;
								Minutos[j].rConsumo1min			:= Minutos[j].rConsumo1min + EstruturaBancoMinuto[i].rConsumo1min;
								Minutos[j].rDemanda1min 		:= Minutos[j].rDemanda1min + EstruturaBancoMinuto[i].rDemanda1min;
								Minutos[j].rFatorDePotencia1min := Minutos[j].rFatorDePotencia1min + EstruturaBancoMinuto[i].rFatorDePotencia1min;
								Minutos[j].Timestamp 			:= EstruturaBancoMinuto[i].Timestamp;
							END_IF
						END_FOR
					END_FOR
					
					iEstadoLeitura			:= 4;
				END_IF
			END_IF
		END_IF
		
		
		IF xDiaSelecionado THEN
			//Le os 15 minutos
			stPara2.eParaType	:= E_ExpParameterType.Float32;
			stPara2.nParaSize	:= SIZEOF(TagAProcurar);
			stPara2.sParaName	:= 'rMedia15min';
			
			IF sMedidor = '' THEN
				sMedidor := '1';
			END_IF
			
			arString[0] := 'SELECT * FROM dbexcelsior.media15min WHERE medidor in (';
			arString[1] := sMedidor;
			arString[2] := ') AND timestamps BETWEEN ';
			arString[3] := CONCAT(CONCAT('("',LEFT(STR:=RIGHT(STR:= DT_TO_STRING(Timestamp - T#3H), SIZE:= 19) , SIZE:= 10)),'-00:00:00")');
			arString[4] := ' AND ';
			arString[5] := CONCAT(CONCAT('("',	RIGHT(STR:= DT_TO_STRING(Timestamp - T#3H), SIZE:= 19)), '");');
			
			CONCAT2(pSrcString1:= ADR(arString[0]), pSrcString2:= ADR(arString[1]), pDstString:= ADR(arString[6]), nDstSize:= SIZEOF(arString[6]));
			CONCAT2(pSrcString1:= ADR(arString[6]), pSrcString2:= ADR(arString[2]), pDstString:= ADR(arString[7]), nDstSize:= SIZEOF(arString[7]));
			CONCAT2(pSrcString1:= ADR(arString[7]), pSrcString2:= ADR(arString[3]), pDstString:= ADR(arString[8]), nDstSize:= SIZEOF(arString[8]));
			CONCAT2(pSrcString1:= ADR(arString[8]), pSrcString2:= ADR(arString[4]), pDstString:= ADR(arString[9]), nDstSize:= SIZEOF(arString[9]));
			CONCAT2(pSrcString1:= ADR(arString[9]), pSrcString2:= ADR(arString[5]), pDstString:= ADR(arString[10]), nDstSize:= SIZEOF(arString[10]));
			
			sCmdEscreve2 := arString[10];
			
			//limpa o array
			FOR i := 1 TO 96 DO
				Media15Min[i].Medidor := 0;
				Media15Min[i].rMedia15min := 0;
				Media15Min[i].rConsumo15min := 0;
				Media15Min[i].rFatorDePotencia15min := 0;
				Media15Min[i].Timestamp := DT#1970-1-1-0:0:0;
			END_FOR
			
			// call functionblock
			IF fbPLCDBCmd2.ExecuteDataReturn
				(
					hDBID := 1,
						pExpression := ADR(sCmdEscreve2),
						cbExpression := SIZEOF(sCmdEscreve2),
						pData := ADR(TagAProcurar),
						cbData := SIZEOF(TagAProcurar),
						pParameter := ADR(stPara2),
						cbParameter := SIZEOF(stPara2),
						nStartIndex := 0,
						nRecordCount := 5760,
						pReturnData := ADR(EstruturaBancoMedia15min),
						cbReturnData := SIZEOF(EstruturaBancoMedia15min),
						pRecords := ADR(nRecords))
			THEN
				IF fbPLCDBCmd2.bError THEN
					sMensagemErro := 'Nao conseguiu a tag';
				ELSE
					sMensagemErro	:= 'Conseguiu a tag';
					iEstadoLeitura			:= 4;
	
					
					FOR i := 1 TO 5760 DO
						IF EstruturaBancoMedia15min[i].Timestamp <> DT#1970-1-1-0:0:0 THEN
							times := DT_TO_SYSTEMTIME(EstruturaBancoMedia15min[i].Timestamp);
							posicao := PosicaoAtualdos15[times.wHour,times.wMinute];
							Media15Min[posicao].rMedia15min				:= Media15Min[posicao].rMedia15min + EstruturaBancoMedia15min[i].rMedia15min;
							Media15Min[posicao].rFatorDePotencia15min	:= Media15Min[posicao].rFatorDePotencia15min + EstruturaBancoMedia15min[i].rFatorDePotencia15min;
							Media15Min[posicao].rConsumo15min			:= Media15Min[posicao].rConsumo15min + EstruturaBancoMedia15min[i].rConsumo15min;
							Media15Min[posicao].Timestamp				:= EstruturaBancoMedia15min[i].Timestamp;
							Media15Min[posicao].Medidor					:= EstruturaBancoMedia15min[i].Medidor;
						END_IF
					END_FOR
				END_IF
			END_IF
		END_IF
		
		
		IF xMesSelecionado THEN
			//Le os dias
			stPara2.eParaType	:= E_ExpParameterType.Float32;
			stPara2.nParaSize	:= SIZEOF(TagAProcurar);
			stPara2.sParaName	:= 'rMediaDia';
			
			arString[0] := 'SELECT * FROM dbexcelsior.mediadia WHERE medidor in (';
			arString[1] := sMedidor;
			arString[2] := ') AND timestamps BETWEEN ';
			arString[3] := CONCAT(CONCAT('("',	LEFT(STR:= RIGHT(STR:= DT_TO_STRING(Timestamp - T#3H), SIZE:= 19), SIZE:= 7)),'-01-00:00:00")');
			arString[4] := ' AND ';
			arString[5] := CONCAT(CONCAT('("',	LEFT(STR:= RIGHT(STR:= DT_TO_STRING(Timestamp - T#3H), SIZE:= 19), SIZE:= 7)),'-01-23:59:59" + INTERVAL 1 MONTH - INTERVAL 1 DAY);');
			
			CONCAT2(pSrcString1:= ADR(arString[0]), pSrcString2:= ADR(arString[1]), pDstString:= ADR(arString[6]), nDstSize:= SIZEOF(arString[6]));
			CONCAT2(pSrcString1:= ADR(arString[6]), pSrcString2:= ADR(arString[2]), pDstString:= ADR(arString[7]), nDstSize:= SIZEOF(arString[7]));
			CONCAT2(pSrcString1:= ADR(arString[7]), pSrcString2:= ADR(arString[3]), pDstString:= ADR(arString[8]), nDstSize:= SIZEOF(arString[8]));
			CONCAT2(pSrcString1:= ADR(arString[8]), pSrcString2:= ADR(arString[4]), pDstString:= ADR(arString[9]), nDstSize:= SIZEOF(arString[9]));
			CONCAT2(pSrcString1:= ADR(arString[9]), pSrcString2:= ADR(arString[5]), pDstString:= ADR(arString[10]), nDstSize:= SIZEOF(arString[10]));
			
			sCmdEscreve3 := arString[10];
			
			//limpa o array
			FOR i := 1 TO 31 DO
				MediaDia[i].Medidor := 0;
				MediaDia[i].rMediaDia := 0;
				MediaDia[i].rConsumoDia := 0;
				MediaDia[i].rFatorDePotenciaDia := 0;
				MediaDia[i].Timestamp := DT#1970-1-1-0:0:0;
			END_FOR
			
			
			// call functionblock
			IF fbPLCDBCmd3.ExecuteDataReturn
				(
					hDBID := 1,
						pExpression := ADR(sCmdEscreve3),
						cbExpression := SIZEOF(sCmdEscreve3),
						pData := ADR(TagAProcurar),
						cbData := SIZEOF(TagAProcurar),
						pParameter := ADR(stPara2),
						cbParameter := SIZEOF(stPara2),
						nStartIndex := 0,
						nRecordCount := 1860,
						pReturnData := ADR(EstruturaBancoMediaDia),
						cbReturnData := SIZEOF(EstruturaBancoMediaDia),
						pRecords := ADR(nRecords))
			THEN
				IF fbPLCDBCmd3.bError THEN
					sMensagemErro := 'Nao conseguiu a tag';
				ELSE
					sMensagemErro := 'Conseguiu a tag';
					iEstadoLeitura			:= 4;
	
					
					FOR i := 1 TO 1860 DO
							times := DT_TO_SYSTEMTIME(EstruturaBancoMediaDia[i].Timestamp);
							
							IF (EstruturaBancoMediaDia[i].Timestamp <> DT#1970-1-1-00:00:00) THEN
								MediaDia[times.wDay].rMediaDia				:= MediaDia[times.wDay].rMediaDia + EstruturaBancoMediaDia[i].rMediaDia;
								MediaDia[times.wDay].rFatorDePotenciaDia	:= MediaDia[times.wDay].rFatorDePotenciaDia + EstruturaBancoMediaDia[i].rFatorDePotenciaDia;
								MediaDia[times.wDay].rConsumoDia			:= MediaDia[times.wDay].rConsumoDia + EstruturaBancoMediaDia[i].rConsumoDia;
								MediaDia[times.wDay].Timestamp				:= EstruturaBancoMediaDia[i].Timestamp;
								MediaDia[times.wDay].Medidor				:= EstruturaBancoMediaDia[i].Medidor;
							END_IF
					END_FOR
				END_IF
			END_IF
		END_IF
		
		IF xAnoSelecionado THEN
			//Le os meses
			stPara2.eParaType	:= E_ExpParameterType.Float32;
			stPara2.nParaSize	:= SIZEOF(TagAProcurar);
			stPara2.sParaName	:= 'rMediaMes';
			
			arString[0] := 'SELECT * FROM dbexcelsior.mediames WHERE medidor in (';
			arString[1] := sMedidor;
			arString[2] := ') AND timestamps BETWEEN ';
			arString[3] := CONCAT(CONCAT('("',	LEFT(STR:= RIGHT(STR:= DT_TO_STRING(Timestamp - T#3H), SIZE:= 19), SIZE:= 4)),'-01-01-00:00:00")');
			arString[4] := ' AND ';
			arString[5] := CONCAT(CONCAT('("',	LEFT(STR:= RIGHT(STR:= DT_TO_STRING(Timestamp - T#3H), SIZE:= 19), SIZE:= 4)),'-12-31-23:59:59");');
			
			CONCAT2(pSrcString1:= ADR(arString[0]), pSrcString2:= ADR(arString[1]), pDstString:= ADR(arString[6]), nDstSize:= SIZEOF(arString[6]));
			CONCAT2(pSrcString1:= ADR(arString[6]), pSrcString2:= ADR(arString[2]), pDstString:= ADR(arString[7]), nDstSize:= SIZEOF(arString[7]));
			CONCAT2(pSrcString1:= ADR(arString[7]), pSrcString2:= ADR(arString[3]), pDstString:= ADR(arString[8]), nDstSize:= SIZEOF(arString[8]));
			CONCAT2(pSrcString1:= ADR(arString[8]), pSrcString2:= ADR(arString[4]), pDstString:= ADR(arString[9]), nDstSize:= SIZEOF(arString[9]));
			CONCAT2(pSrcString1:= ADR(arString[9]), pSrcString2:= ADR(arString[5]), pDstString:= ADR(arString[10]), nDstSize:= SIZEOF(arString[10]));
			
			sCmdEscreve4 := arString[10];
			
			//limpa o array
			FOR i := 1 TO 12 DO
				MediaMes[i].Medidor := 0;
				MediaMes[i].rMediaMes := 0;
				MediaMes[i].rConsumoMes := 0;
				MediaMes[i].rFatorDePotenciaMes := 0;
				MediaMes[i].Timestamp := DT#1970-1-1-0:0:0;
			END_FOR
			
			// call functionblock
			IF fbPLCDBCmd4.ExecuteDataReturn
				(
					hDBID := 1,
						pExpression := ADR(sCmdEscreve4),
						cbExpression := SIZEOF(sCmdEscreve4),
						pData := ADR(TagAProcurar),
						cbData := SIZEOF(TagAProcurar),
						pParameter := ADR(stPara2),
						cbParameter := SIZEOF(stPara2),
						nStartIndex := 0,
						nRecordCount := 720,
						pReturnData := ADR(EstruturaBancoMediaMes),
						cbReturnData := SIZEOF(EstruturaBancoMediaMes),
						pRecords := ADR(nRecords))
			THEN
				IF fbPLCDBCmd4.bError THEN
					sMensagemErro := 'Nao conseguiu a tag';
				ELSE
					sMensagemErro	:= 'Conseguiu a tag';
					iEstadoLeitura			:= 4;
	
					
					FOR i := 1 TO 720 DO
						times 										:= DT_TO_SYSTEMTIME(EstruturaBancoMediaMes[i].Timestamp);
						
						IF (EstruturaBancoMediaMes[i].Timestamp <> DT#1970-1-1-00:00:00) THEN
							MediaMes[times.wMonth].rMediaMes			:= MediaMes[times.wMonth].rMediaMes+EstruturaBancoMediaMes[i].rMediaMes;
							MediaMes[times.wMonth].rFatorDePotenciaMes	:= MediaMes[times.wMonth].rFatorDePotenciaMes+EstruturaBancoMediaMes[i].rFatorDePotenciaMes;
							MediaMes[times.wMonth].rConsumoMes			:= MediaMes[times.wMonth].rConsumoMes+EstruturaBancoMediaMes[i].rConsumoMes;
							MediaMes[times.wMonth].Timestamp			:= EstruturaBancoMediaMes[i].Timestamp;
							MediaMes[times.wMonth].Medidor				:= EstruturaBancoMediaMes[i].Medidor;
						END_IF
					END_FOR
				END_IF
			END_IF
		END_IF

	4: // FechaConexao conexao
		IF fbSQLDatabase2.Disconnect() THEN

			xAtualizaInterno	:= FALSE;
			xAtualiza			:= FALSE;
			xTerminouLeitura	:= TRUE;
			
			IF fbSQLDatabase2.bError THEN
				iEstadoLeitura := 1;
			ELSE
				iEstadoLeitura := 1;
			END_IF
		END_IF
END_CASE
END_ACTION

END_FUNCTION_BLOCK

// FBs/MedicaoEnergia/FB_DBCentroDeCustos
FUNCTION_BLOCK FB_DBCentroDeCustos
VAR_IN_OUT
	CentrosDeCustos		: ARRAY[*] OF stCentroDeCusto;
END_VAR
VAR_INPUT
	xCriaTabelas					: BOOL;				// tenta criar a tabela
	iNumeroDataBase					: INT	:= 1;		// id do database
	sNomeCentroDeCustos				: STRING(255);
	sMedidoresSelecionados			: STRING(1000);
	xLeDadosCentroDeCusto			: BOOL;
	xGravaNovoCentroDeCusto			: BOOL;
	xDeleteCentroDeCustos			: BOOL;
	xLeTodos						: BOOL;
	xDeletaTodos					: BOOL;
	xReset							: BOOL;
END_VAR
VAR_OUTPUT
	xOcupado 				: BOOL;
	xTabelaCriada			: BOOL;
	xTermineiDeLer			: BOOL;
	xTermineiDeEscrever		: BOOL;
	xTermineiDeDeletar		: BOOL;
END_VAR
VAR
	//Cria table
	rtCria				: R_TRIG;
	xComecaCriarTabelas	: BOOL;
	fbPLCDBCreate		: FB_PLCDBCreateEvt(sNetID := '', tTimeout := T#30S);
	
	ColumnInfo : ARRAY[0..2] OF ST_ColumnInfo := [	(sName := 'NomeGrupo',	eType := E_ColumnType.NVarChar,	nLength := 255, sProperty := 'DEFAULT $'-$''),
													(sName := 'MedidoresSelecionados',	eType := E_ColumnType.NVarChar, nLength := 1000, sProperty := 'DEFAULT $'-$''),
													(sName := 'timestamps', 	eType := E_ColumnType.DateTime, nLength := 4, sProperty := 'DEFAULT CURRENT_TIMESTAMP ON UPDATE CURRENT_TIMESTAMP')];
													
			
	//Grava valores
	xEscreve			: BOOL;
	rtEscreve			: R_TRIG;
	fbSqlCommand		: FB_SQLCommandEvt(sNetID := '', tTimeout := T#30S);
	fbSQLDatabase		: FB_SQLDatabaseEvt(sNetID := '', tTimeout := T#30S);
	//arStringConcat		: ARRAY[1..60] OF STRING(255);
	//arSplit				: ARRAY[1.54] OF STRING(255); 
	sCmdParte1			: STRING(1000);
	sCmdParte2			: STRING(1000);
	sCmd1				: STRING(255);
	sCmd2				: STRING(255);
	sCmd3				: STRING(255);
	sMensagemErro1 		: STRING;
	xAberto 			: BOOL;
	rtComecaEscrever 	: R_TRIG;
	iEstado 			: INT := 1;
	i					: INT;
	
	
		
	//Le Valores
	sCmdEscreve					: STRING(1000);
	sMensagemErro2				: STRING;
	EstruturaBancoGrupos		: ARRAY[1..150] OF stCentroDeCusto;
	nRecords					: UDINT;
	TagAProcurar				: STRING;
	diCima						: DINT;
	diBaixo						: DINT;
	iEstadoLeitura				: INT := 1;
	j							: INT;
	stPara						: ST_ExpParameter;
	fbSQLDatabase2				: FB_SQLDatabaseEvt(sNetID := '', tTimeout := T#30S);
	fbPLCDBCmd					: FB_PLCDBCmdEvt(sNetID := '', tTimeout := T#30S);
	arString2					: ARRAY[0..6] OF STRING(255);
	rtLeitura					: R_TRIG;
	xAtualizaInterno			: BOOL;
	
	
	
	
	//Deleta Valores
	xDelete				: BOOL;
	rtDelete			: R_TRIG;
	fbSqlCommand1		: FB_SQLCommandEvt(sNetID := '', tTimeout := T#30S);
	fbSQLDatabase3		: FB_SQLDatabaseEvt(sNetID := '', tTimeout := T#30S);
	sCmdDelete			: STRING(255);
	sMensagemErro3 		: STRING;
	xAbertoDelete 		: BOOL;
	rtComecaDelte 		: R_TRIG;
	iEstadoDelete 		: INT := 1;
	rtReset				: R_TRIG;
END_VAR


IF xLicensaValida651641iih THEN
	GeraTabela();
	rtEscreve(CLK:= xGravaNovoCentroDeCusto, Q=> );
	rtLeitura(CLK:= xLeDadosCentroDeCusto, Q=> );
	rtDelete(CLK:= xDeleteCentroDeCustos, Q=> );
	rtReset(CLK:= xReset, Q=> );
	
	
	IF rtReset.Q THEN
	xTermineiDeLer			:= FALSE;
	xTermineiDeDeletar		:= FALSE;
	xTermineiDeEscrever 	:= FALSE;
	END_IF
	
	IF rtEscreve.Q THEN
	xEscreve := TRUE;
	xTermineiDeEscrever := FALSE;
	END_IF
	
	IF rtLeitura.Q THEN
	xAtualizaInterno := TRUE;
	END_IF
	
	IF rtDelete.Q THEN
	xDelete := TRUE;
	END_IF
	
	LeValores();
	GravaValores();
	DeleteValores();	
END_IF;

ACTION DeleteValores:

CASE iEstadoDelete OF
	1: //Esperando
		IF xDelete THEN
			IF xAbertoDelete THEN
				iEstadoDelete := 3;	//Caso para abrir a conexão
				xTermineiDeDeletar		:= FALSE;
			ELSE
				iEstadoDelete := 2;	//Caso em que a conexão já foi aberta
			END_IF
		END_IF
		
	2: //abre conexao
		IF fbSQLDatabase3.Connect(INT_TO_UDINT(iNumeroDataBase)) THEN
			IF fbSQLDatabase3.bError THEN
				IF fbSQLDatabase3.ipTcResult.nEventId = 1828 THEN
					// se der isso ele nao fica tentando e gerando uma caralhada de erro pq nao tem a lisença
					iEstadoDelete := 0;
				ELSE
					iEstadoDelete := 2;
				END_IF
			ELSE
				IF fbSQLDatabase3.bConnected THEN
					iEstadoDelete := 3;
					xAbertoDelete := TRUE;
				ELSE
					iEstadoDelete := 5;
					xAbertoDelete := FALSE;
				END_IF
			END_IF
		END_IF
		
	3:
		IF fbSQLDatabase3.CreateCmd(ADR(fbSqlCommand1)) THEN
			IF fbSQLDatabase3.bError THEN
				iEstadoDelete := 3;
			ELSE
				iEstadoDelete := 4;
			END_IF
		END_IF
		
	4: // le o role
		IF (xDeletaTodos) THEN
			sCmdDelete := 'DELETE FROM dbexcelsior.centrodecustos';
		ELSE
			sCmdDelete := CONCAT(CONCAT('DELETE FROM dbexcelsior.centrodecustos WHERE NomeGrupo="',sNomeCentroDeCustos),'";');
		END_IF

	
		IF fbSqlCommand1.Execute(pSQLCmd := ADR(sCmdDelete), cbSQLCmd := SIZEOF(sCmdDelete)) THEN
			IF fbSqlCommand1.bError THEN
				IF fbSqlCommand1.ipTcResult.nEventId = 61 THEN
				// Esse erro acontece quando o database não tá criado, nesse caso ele tenta criar
					iEstadoDelete := 1;
					xCriaTabelas := TRUE;
				ELSE
					iEstadoDelete := 2;
				END_IF
				sMensagemErro3 := 'Nao conseguiu a tag';
			ELSE
				sMensagemErro3	:= 'Conseguiu a tag';
			END_IF
			iEstadoDelete := 5;
			xDelete					:= FALSE;
			xDeleteCentroDeCustos 	:= FALSE;
			xTermineiDeDeletar		:= TRUE;
		END_IF
		
		
	5: // FechaConexao conexao
			IF fbSQLDatabase3.Disconnect() THEN
	
				xDeleteCentroDeCustos		:= FALSE;
				xDelete					:= FALSE;
	
				IF fbSQLDatabase3.bError THEN
					iEstadoDelete := 1;
				ELSE
					iEstadoDelete := 1;
					xAbertoDelete := FALSE;
				END_IF
			END_IF
END_CASE
END_ACTION

ACTION GeraTabela:

rtCria(CLK := xCriaTabelas, Q =>);

IF rtCria.q THEN
	xComecaCriarTabelas		:= TRUE;
	xOcupado				:= TRUE;
END_IF

IF xComecaCriarTabelas THEN
		//Cria a tabela com os minutos inidividuais de cada um dos 15 min
		IF fbPLCDBCreate.Table
			(
				hDBID := INT_TO_UDINT(iNumeroDataBase),
					sTableName := 'centrodecustos',
					pTableCfg := ADR(ColumnInfo),
					cbTableCfg := SIZEOF(ColumnInfo))
		THEN
			IF NOT fbPLCDBCreate.bError  OR (fbPLCDBCreate.bError AND fbPLCDBCreate.ipTcResult.nEventId = 60) THEN
				xTabelaCriada := TRUE;
			ELSE
				xTabelaCriada := FALSE;
			END_IF
		END_IF
	
	IF (xTabelaCriada) THEN
		xComecaCriarTabelas		:= FALSE;
		xCriaTabelas	:= FALSE;
		xOcupado := FALSE;
	ELSE
		xCriaTabelas	:= FALSE;
		xComecaCriarTabelas		:= FALSE;
		xOcupado := FALSE;
	END_IF 
	
ELSE
	xOcupado := FALSE;
END_IF
END_ACTION

ACTION GravaValores:

CASE iEstado OF
	1: //Esperando
		IF xEscreve THEN
			IF xAberto THEN
				iEstado := 3;	//Caso para abrir a conexão
				xTermineiDeEscrever		:= FALSE;
			ELSE
				iEstado := 2;	//Caso em que a conexão já foi aberta
			END_IF
		END_IF
		
	2: //abre conexao
		IF fbSqlDatabase.Connect(int_to_udint(iNumeroDataBase)) THEN
			IF fbSqlDatabase.bError THEN
				IF fbSqlDatabase.ipTcResult.nEventId = 1828 THEN
					// se der isso ele nao fica tentando e gerando uma caralhada de erro pq nao tem a lisença
					iEstado := 0;
				ELSE
					iEstado := 2;
				END_IF
			ELSE
				IF fbSqlDatabase.bConnected THEN
					iEstado := 3;
					xAberto := TRUE;
				ELSE
					iEstado := 5;
					xAberto := FALSE;
				END_IF
			END_IF
		END_IF
		
	3:
		IF fbSqlDatabase.CreateCmd(ADR(fbSqlCommand)) THEN
			IF fbSqlDatabase.bError THEN
				iEstado := 3;
			ELSE
				iEstado := 4;
			END_IF
		END_IF
		
		4: // le o role
		//'INSERT INTO dbexcelsior.centrodecustos(NomeGrupo,MedidoresSelecionados) VALUES (sNomeCentroDeCustos, sMedidoresSelecionados);'	
		IF sNomeCentroDeCustos = ''THEN
			sNomeCentroDeCustos := 'Failed';
		END_IF
		//sCmd	:= CONCAT(CONCAT(CONCAT(CONCAT('INSERT INTO dbexcelsior.centrodecustos(NomeGrupo,MedidoresSelecionados) VALUES ("',sNomeCentroDeCustos),'","'),sMedidoresSelecionados),'");');
		sCmd1	:= 'INSERT INTO dbexcelsior.centrodecustos(NomeGrupo,MedidoresSelecionados) VALUES ("';
		sCmd2	:= CONCAT(sNomeCentroDeCustos, '","');
		CONCAT2(pSrcString1:= ADR(sCmd1), pSrcString2:= ADR(sCmd2), pDstString:= ADR(sCmdParte1), nDstSize:= 1000);
		
		sCmd3	:= CONCAT(sMedidoresSelecionados, '");');
		CONCAT2(pSrcString1:= ADR(sCmdParte1), pSrcString2:= ADR(sCmd3), pDstString:= ADR(sCmdParte2), nDstSize:= 1000);
		
		IF fbSQLCommand.Execute(pSQLCmd := ADR(sCmdParte2), cbSQLCmd := SIZEOF(sCmdParte2)) THEN
			IF fbSQLCommand.bError THEN
				IF fbSQLCommand.ipTcResult.nEventId = 61 THEN
				// Esse erro acontece quando o database não tá criado, nesse caso ele tenta criar
				iEstado := 1;
					xCriaTabelas := TRUE;
				ELSE
					iEstado := 2;
				END_IF
				sMensagemErro1 := 'Nao conseguiu a tag';
			ELSE
				sMensagemErro1	:= 'Conseguiu a tag';
			END_IF
			iEstado := 5;
			xEscreve				:= FALSE;
			xGravaNovoCentroDeCusto := FALSE;
			xTermineiDeEscrever		:= TRUE;
		END_IF
		
		
	5: // FechaConexao conexao
			IF fbSqlDatabase.Disconnect() THEN
	
				xGravaNovoCentroDeCusto		:= FALSE;
				xEscreve					:= FALSE;
	
				IF fbSqlDatabase.bError THEN
					iEstado := 1;
				ELSE
					iEstado := 1;
					xAberto := FALSE;
				END_IF
			END_IF
END_CASE
END_ACTION

ACTION LeValores:
CASE iEstadoLeitura OF
	1: //Esperando
		IF xAtualizaInterno THEN
			xTermineiDeLer := FALSE;
			iEstadoLeitura := 2;
		END_IF

	2: //abre conexao
		IF fbSQLDatabase2.Connect(INT_TO_UDINT(iNumeroDataBase)) THEN
			IF fbSQLDatabase2.bError THEN
				IF fbSQLDatabase2.ipTcResult.ipSourceInfo.sName = 'ADSERR_DEVICE_LICENSENOTFOUND' THEN
					// se der isso ele nao fica tentando e gerando uma caralhada de erro pq nao tem a lisença
					iEstadoLeitura := 0;
				ELSE
					iEstadoLeitura := 2;
				END_IF
			ELSE
				IF fbSQLDatabase2.bConnected THEN
					iEstadoLeitura := 3;
				END_IF
			END_IF
		END_IF

	3: // Le os DADOS
		stPara.eParaType	:= E_ExpParameterType.STRING_;
		stPara.nParaSize	:= SIZEOF(TagAProcurar);
		stPara.sParaName	:= 'NomeGrupo';

		
		//RECUPERANDO DADOS DOS MINUTOS
		diBaixo	:= LOWER_BOUND(CentrosDeCustos, 1);
		diCima	:= UPPER_BOUND(CentrosDeCustos, 1);
		
		
		IF (xLeTodos) THEN
			sCmdEscreve := 'SELECT * FROM dbexcelsior.centrodecustos;';
		ELSE
			sCmdEscreve := CONCAT(CONCAT('SELECT * FROM dbexcelsior.centrodecustos WHERE NomeGrupo="',sNomeCentroDeCustos),'";');
		END_IF

		
		// call functionblock
		IF fbPLCDBCmd.ExecuteDataReturn
			(
				hDBID := 1,
					pExpression := ADR(sCmdEscreve),
					cbExpression := SIZEOF(sCmdEscreve),
					pData := ADR(TagAProcurar),
					cbData := SIZEOF(TagAProcurar),
					pParameter := ADR(stPara),
					cbParameter := SIZEOF(stPara),
					nStartIndex := 0,
					nRecordCount := DINT_TO_UDINT(diCima),
					pReturnData := ADR(EstruturaBancoGrupos),
					cbReturnData := SIZEOF(EstruturaBancoGrupos),
					pRecords := ADR(nRecords))
		THEN
			IF fbPLCDBCmd.bError THEN
				sMensagemErro2 := 'Nao conseguiu a tag';
			ELSE
				sMensagemErro2	:= 'Conseguiu a tag';
				iEstadoLeitura			:= 4;

				FOR j := TO_INT(diBaixo) TO TO_INT(diCima) DO
					CentrosDeCustos[j].MedidoresSelecionados		:= EstruturaBancoGrupos[j].MedidoresSelecionados;
					CentrosDeCustos[j].NomeGrupo					:= EstruturaBancoGrupos[j].NomeGrupo;
					CentrosDeCustos[j].Timestamp					:= EstruturaBancoGrupos[j].Timestamp;
					xTermineiDeLer := TRUE;
				END_FOR

			END_IF
		ELSE
			xTermineiDeLer := FALSE;
		END_IF

	4: // FechaConexao conexao
		IF fbSQLDatabase2.Disconnect() THEN

			xAtualizaInterno		:= FALSE;
			xLeDadosCentroDeCusto	:= FALSE;
			
			IF fbSQLDatabase2.bError THEN
				iEstadoLeitura := 1;
			ELSE
				iEstadoLeitura := 1;
			END_IF
		END_IF
END_CASE
END_ACTION

END_FUNCTION_BLOCK

// FBs/MedicaoEnergia/FB_DBMedidores
//{attribute 'hide_all_locals'}
FUNCTION_BLOCK FB_DBMedidores
VAR_IN_OUT
	Minutos				: ARRAY[*] OF stMinuto;
	Media15Min			: ARRAY[*] OF stMedia15min;
	MediaDia			: ARRAY[*] OF stMediaDia;
	MediaMes			: ARRAY[*] OF stMediaMes;
	PosicaoAtualdos15	: ARRAY[*,*] OF INT;
END_VAR
VAR_INPUT
	xCriaTabelas			: BOOL;				// tenta criar a tabela
	iNumeroDataBase			: INT	:= 1;		// id do database
	iMedidor				: INT;
	xMedidorOnline			: BOOL;
	rDemanda1min			: REAL;
	rFP1min					: REAL;
	rConsumo1min			: REAL;
	xEscreveMinuto			: BOOL;
	Timestamp				: DT;
	xAtualiza				: BOOL;
	x15minSelecionado		: BOOL;
	xDiaSelecionado			: BOOL;
	xMesSelecionado			: BOOL;
	xAnoSelecionado			: BOOL;
END_VAR
VAR_OUTPUT
	xOcupado 				: BOOL;
	xTodasTabelasCriadas	: BOOL;
	xTerminouLeitura		: BOOL := FALSE;
END_VAR
VAR		
	
	//Cria table
	rtCria				: R_TRIG;
	xComecaCriarTabelas	: BOOL;
	xTabela1Criada		: BOOL;
	xTabela2Criada		: BOOL;
	xTabela3Criada		: BOOL;
	xTabela4Criada		: BOOL;
	xTabela5Criada		: BOOL;
	
	fbPLCDBCreate1	: FB_PLCDBCreateEvt(sNetID := '', tTimeout := T#30S);
	fbPLCDBCreate2	: FB_PLCDBCreateEvt(sNetID := '', tTimeout := T#30S);
	fbPLCDBCreate3	: FB_PLCDBCreateEvt(sNetID := '', tTimeout := T#30S);
	fbPLCDBCreate4	: FB_PLCDBCreateEvt(sNetID := '', tTimeout := T#30S);
	fbPLCDBCreate5	: FB_PLCDBCreateEvt(sNetID := '', tTimeout := T#30S);
	
	ColumnInfo1 : ARRAY[0..4] OF ST_ColumnInfo := [	(sName := 'rDemanda1min',	eType := E_ColumnType.REAL_,	nLength := 4),
													(sName := 'rFatorDePotencia1min',	eType := E_ColumnType.REAL_,	nLength := 4),
													(sName := 'rConsumo1min',	eType := E_ColumnType.REAL_,	nLength := 4),
													(sName := 'medidor',	eType := E_ColumnType.Integer, 	nLength := 2),
													(sName := 'timestamps', 	eType := E_ColumnType.DateTime, nLength := 4, sProperty := 'DEFAULT CURRENT_TIMESTAMP ON UPDATE CURRENT_TIMESTAMP')];
													
	ColumnInfo2 : ARRAY[0..4] OF ST_ColumnInfo := [	(sName := 'rMedia15min',eType := E_ColumnType.REAL_,	nLength := 4),
													(sName := 'rFatorDePotencia15min',	eType := E_ColumnType.REAL_,	nLength := 4),
													(sName := 'rConsumo15min',	eType := E_ColumnType.REAL_,	nLength := 4),
													(sName := 'medidor',	eType := E_ColumnType.Integer, 	nLength := 2),
													(sName := 'timestamps', 	eType := E_ColumnType.DateTime, nLength := 4, sProperty := 'DEFAULT CURRENT_TIMESTAMP ON UPDATE CURRENT_TIMESTAMP')];
													
	ColumnInfo3 : ARRAY[0..4] OF ST_ColumnInfo := [	(sName := 'rMediaDia',	eType := E_ColumnType.REAL_,	nLength := 4),
													(sName := 'rFatorDePotenciaDia',	eType := E_ColumnType.REAL_,	nLength := 4),
													(sName := 'rConsumoDia',	eType := E_ColumnType.REAL_,	nLength := 4),
													(sName := 'medidor',	eType := E_ColumnType.Integer, 	nLength := 2),
													(sName := 'timestamps', 	eType := E_ColumnType.DateTime, nLength := 4, sProperty := 'DEFAULT CURRENT_TIMESTAMP ON UPDATE CURRENT_TIMESTAMP')];
													
													
	ColumnInfo4 : ARRAY[0..4] OF ST_ColumnInfo := [	(sName := 'rMediaMes',	eType := E_ColumnType.REAL_,	nLength := 4),
													(sName := 'rFatorDePotenciaMes',	eType := E_ColumnType.REAL_,	nLength := 4),
													(sName := 'rConsumoMes',	eType := E_ColumnType.REAL_,	nLength := 4),
													(sName := 'medidor',	eType := E_ColumnType.Integer, 	nLength := 2),
													(sName := 'timestamps', 	eType := E_ColumnType.DateTime, nLength := 4, sProperty := 'DEFAULT CURRENT_TIMESTAMP ON UPDATE CURRENT_TIMESTAMP')];

	ColumnInfo5 : ARRAY[0..4] OF ST_ColumnInfo := [	(sName := 'rMediaAno',	eType := E_ColumnType.REAL_,	nLength := 4),
													(sName := 'rFatorDePotenciaAno',	eType := E_ColumnType.REAL_,	nLength := 4),
													(sName := 'rConsumoAno',	eType := E_ColumnType.REAL_,	nLength := 4),
													(sName := 'medidor',	eType := E_ColumnType.Integer, 	nLength := 2),
													(sName := 'timestamps', 	eType := E_ColumnType.DateTime, nLength := 4, sProperty := 'DEFAULT CURRENT_TIMESTAMP ON UPDATE CURRENT_TIMESTAMP')];
													
	//Grava valores
	xEscreve			: BOOL;
	rtEscreve			: R_TRIG;
	tonEscrita			: TON;
	arString			: ARRAY[0..5] OF STRING(255);
	fbSqlCommand		: FB_SQLCommandEvt(sNetID := '', tTimeout := T#30S);
	fbSQLDatabase		: FB_SQLDatabaseEvt(sNetID := '', tTimeout := T#30S);
	sCmd				: STRING(1000);
	sMensagemErro1 		: STRING;
	xAberto 			: BOOL;
	rtComecaEscrever 	: R_TRIG;
	iEstado 			: INT := 1;
	i					: INT;
	
	//Le Valores
	sCmdEscreve1				: STRING(1000);
	sCmdEscreve2				: STRING(1000);
	sCmdEscreve3				: STRING(1000);
	sCmdEscreve4				: STRING(1000);
	sMensagemErro2				: STRING;
	EstruturaBancoMinuto		: ARRAY[1..15] OF stMinuto;
	EstruturaBancoMedia15min	: ARRAY[1..96] OF stMedia15min;
	EstruturaBancoMediaDia		: ARRAY[1..31] OF stMediaDia;
	EstruturaBancoMediaMes		: ARRAY[1..12] OF stMediaMes;
	nRecords					: UDINT;
	TagAProcurar				: REAL;
	diCima						: DINT;
	diBaixo						: DINT;
	iEstadoLeitura				: INT := 1;
	j							: INT;
	stPara						: ST_ExpParameter;
	fbSQLDatabase2				: FB_SQLDatabaseEvt(sNetID := '', tTimeout := T#30S);
	fbPLCDBCmd1					: FB_PLCDBCmdEvt(sNetID := '', tTimeout := T#30S);
	fbPLCDBCmd2					: FB_PLCDBCmdEvt(sNetID := '', tTimeout := T#30S);
	fbPLCDBCmd3					: FB_PLCDBCmdEvt(sNetID := '', tTimeout := T#30S);
	fbPLCDBCmd4					: FB_PLCDBCmdEvt(sNetID := '', tTimeout := T#30S);
	arString2					: ARRAY[0..6] OF STRING(255);
	MinutosAtuais				: ARRAY[1..15] OF INT;
	posicao						: INT := 1;
	minute						: TIMESTRUCT;
	times						: TIMESTRUCT;
	rtLeitura1					: R_TRIG;
	rtLeitura2					: R_TRIG;
	rtLeitura3					: R_TRIG;
	rtLeitura4					: R_TRIG;
	rtLeitura5					: R_TRIG;
	xAtualizaInterno			: BOOL;
END_VAR

//Criado Por Augusto Cazzanelli para o Projeto Excelsior
IF xLicensaValida651641iih THEN
	GeraTabela();
	
	rtEscreve(CLK:= xEscreveMinuto, Q=> );
	rtLeitura1(CLK:= xAtualiza, Q=> );
	rtLeitura2(CLK:= x15minSelecionado, Q=> );
	rtLeitura3(CLK:= xDiaSelecionado, Q=> );
	rtLeitura4(CLK:= xMesSelecionado, Q=> );
	rtLeitura5(CLK:= xAnoSelecionado, Q=> );
	
	IF rtLeitura1.Q OR rtLeitura2.Q OR rtLeitura3.Q OR rtLeitura4.Q OR rtLeitura5.Q THEN
		xAtualizaInterno 	:= TRUE;
		xTerminouLeitura	:= FALSE;
	END_IF
	
	
	IF rtEscreve.Q THEN
		xEscreve := TRUE;

	END_IF
	
	GravaValores();
	LeValores();

END_IF;

ACTION GeraTabela:

rtCria(CLK := xCriaTabelas, Q =>);

IF rtCria.q THEN
	xComecaCriarTabelas		:= TRUE;
	xOcupado				:= TRUE;
END_IF

IF xComecaCriarTabelas THEN
		//Cria a tabela com os minutos inidividuais de cada um dos 15 min
		IF fbPLCDBCreate1.Table
			(
				hDBID := INT_TO_UDINT(iNumeroDataBase),
					sTableName := 'minutos',
					pTableCfg := ADR(ColumnInfo1),
					cbTableCfg := SIZEOF(ColumnInfo1))
		THEN
			IF NOT fbPLCDBCreate1.bError  OR (fbPLCDBCreate1.bError AND fbPLCDBCreate1.ipTcResult.nEventId = 60) THEN
				xTabela1Criada := TRUE;
			ELSE
				xTabela1Criada := FALSE;
			END_IF
		END_IF


		//Cria a tabela com a media dos 15 min
		IF fbPLCDBCreate2.Table
		(
				hDBID := INT_TO_UDINT(iNumeroDataBase),
					sTableName := 'media15min',
					pTableCfg := ADR(ColumnInfo2),
					cbTableCfg := SIZEOF(ColumnInfo2))
		THEN
			IF NOT fbPLCDBCreate2.bError  OR (fbPLCDBCreate1.bError AND fbPLCDBCreate2.ipTcResult.nEventId = 60) THEN
				xTabela2Criada := TRUE;
			ELSE
				xTabela2Criada := FALSE;
			END_IF
		END_IF

		//Cria a tabela com a media dos dias
		IF fbPLCDBCreate3.Table
		(
				hDBID := INT_TO_UDINT(iNumeroDataBase),
					sTableName := 'mediadia',
					pTableCfg := ADR(ColumnInfo3),
					cbTableCfg := SIZEOF(ColumnInfo3))
		THEN
			IF NOT fbPLCDBCreate3.bError  OR (fbPLCDBCreate1.bError AND fbPLCDBCreate3.ipTcResult.nEventId = 60) THEN
				xTabela3Criada := TRUE;
			ELSE
				xTabela3Criada := FALSE;
			END_IF
		END_IF	

		//Cria a tabela com a media dos dias para a semana
		IF fbPLCDBCreate4.Table
		(
				hDBID := INT_TO_UDINT(iNumeroDataBase),
					sTableName := 'mediames',
					pTableCfg := ADR(ColumnInfo4),
					cbTableCfg := SIZEOF(ColumnInfo4))
		THEN
			IF NOT fbPLCDBCreate4.bError  OR (fbPLCDBCreate1.bError AND fbPLCDBCreate4.ipTcResult.nEventId = 60) THEN
				xTabela4Criada := TRUE;
			ELSE
				xTabela4Criada := FALSE;
			END_IF
		END_IF
		
		//Cria a tabela com a media do ano
		IF fbPLCDBCreate5.Table
		(
				hDBID := INT_TO_UDINT(iNumeroDataBase),
					sTableName := 'mediaano',
					pTableCfg := ADR(ColumnInfo5),
					cbTableCfg := SIZEOF(ColumnInfo5))
		THEN
			IF NOT fbPLCDBCreate5.bError  OR (fbPLCDBCreate5.bError AND fbPLCDBCreate5.ipTcResult.nEventId = 60) THEN
				xTabela5Criada := TRUE;
			ELSE
				xTabela5Criada := FALSE;
			END_IF
		END_IF



	
	IF (xTabela1Criada AND xTabela2Criada AND xTabela3Criada AND xTabela4Criada AND xTabela4Criada AND xTabela5Criada) THEN
		xComecaCriarTabelas		:= FALSE;
		xCriaTabelas	:= FALSE;
		xTodasTabelasCriadas := TRUE;
		xOcupado := FALSE;
	ELSE
		xCriaTabelas	:= FALSE;
		xComecaCriarTabelas		:= FALSE;
		xTodasTabelasCriadas := FALSE;
		xOcupado := FALSE;
	END_IF 
	
ELSE
	xOcupado := FALSE;
END_IF
END_ACTION

ACTION GravaValores:

CASE iEstado OF
	1: //Esperando
		IF xEscreve AND xMedidorOnline THEN
			IF xAberto THEN
				iEstado := 3;	//Caso para abrir a conexão
			ELSE
				iEstado := 2;	//Caso em que a conexão já foi aberta
			END_IF
		END_IF
		
	2: //abre conexao
		IF fbSqlDatabase.Connect(int_to_udint(iNumeroDataBase)) THEN
			IF fbSqlDatabase.bError THEN
				IF fbSqlDatabase.ipTcResult.nEventId = 1828 THEN
					// se der isso ele nao fica tentando e gerando uma caralhada de erro pq nao tem a lisença
					iEstado := 0;
				ELSE
					iEstado := 2;
				END_IF
			ELSE
				IF fbSqlDatabase.bConnected THEN
					iEstado := 3;
					xAberto := TRUE;
				ELSE
					iEstado := 5;
					xAberto := FALSE;
				END_IF
			END_IF
		END_IF
		
	3:
		IF fbSqlDatabase.CreateCmd(ADR(fbSqlCommand)) THEN
			IF fbSqlDatabase.bError THEN
				iEstado := 3;
			ELSE
				iEstado := 4;
			END_IF
		END_IF
		
		4: // le o role
		//'INSERT INTO dbexcelsior.minutos(rDemanda1min,medidor) VALUES (rDemanda1min, iMedidor);'	
		
		FOR i := 0 TO 3 DO
			arString[i] := '';
		END_FOR
	
		IF xMedidorOnline THEN
			arString[0] := 'INSERT INTO dbexcelsior.minutos(rDemanda1min,rFatorDePotencia1min,rConsumo1min,medidor) VALUES (';
			arString[1] := CONCAT(TO_STRING(rDemanda1min),',');
			arString[2] := CONCAT(TO_STRING(rFP1min),',');
			arString[3] := CONCAT(TO_STRING(rConsumo1min),',');
			arString[4] := CONCAT(TO_STRING(iMedidor),');');
		ELSE
			arString[0] := 'INSERT INTO dbexcelsior.minutos(medidor) VALUE (';
			arString[1] := CONCAT(TO_STRING(iMedidor),');');
			arString[2] := '';
			arString[3] := '';
			arString[4] := '';
		END_IF

	
		sCmd := F_ConcatArray(sArray:= arString);
		
		IF fbSQLCommand.Execute(pSQLCmd := ADR(sCmd), cbSQLCmd := SIZEOF(sCmd)) THEN
			IF fbSQLCommand.bError THEN
				IF fbSQLCommand.ipTcResult.nEventId = 61 THEN
				// Esse erro acontece quando o database não tá criado, nesse caso ele tenta criar
				iEstado := 1;
					xCriaTabelas := TRUE;
				ELSE
					iEstado := 2;
				END_IF
				sMensagemErro1 := 'Nao conseguiu a tag';
			ELSE
				sMensagemErro1	:= 'Conseguiu a tag';
			END_IF
			iEstado := 5;
			xEscreve			:= FALSE;
			xEscreveMinuto := FALSE;
		END_IF
		
		
	5: // FechaConexao conexao
			IF fbSqlDatabase.Disconnect() THEN
	
				xEscreveMinuto		:= FALSE;
				xEscreve			:= FALSE;
	
				IF fbSqlDatabase.bError THEN
					iEstado := 1;
				ELSE
					iEstado := 1;
					xAberto := FALSE;
				END_IF
			END_IF
END_CASE
END_ACTION

ACTION LeValores:
CASE iEstadoLeitura OF
	1: //Esperando
		IF xAtualizaInterno THEN
			iEstadoLeitura := 2;
		END_IF

	2: //abre conexao
		IF fbSQLDatabase2.Connect(INT_TO_UDINT(iNumeroDataBase)) THEN
			IF fbSQLDatabase2.bError THEN
				IF fbSQLDatabase2.ipTcResult.ipSourceInfo.sName = 'ADSERR_DEVICE_LICENSENOTFOUND' THEN
					// se der isso ele nao fica tentando e gerando uma caralhada de erro pq nao tem a lisença
					iEstadoLeitura := 0;
				ELSE
					iEstadoLeitura := 2;
				END_IF
			ELSE
				IF fbSQLDatabase2.bConnected THEN
					iEstadoLeitura := 3;
				END_IF
			END_IF
		END_IF

	3: 
		IF x15minSelecionado THEN
			// Le os Minutos
			stPara.eParaType	:= E_ExpParameterType.Float32;
			stPara.nParaSize	:= SIZEOF(TagAProcurar);
			stPara.sParaName	:= 'rDemanda1min';
	
			
			//RECUPERANDO DADOS DOS MINUTOS
			diBaixo	:= LOWER_BOUND(Minutos, 1);
			diCima	:= UPPER_BOUND(Minutos, 1);
	
			
			arString2[0] := 'SELECT * FROM dbexcelsior.minutos WHERE medidor=';
			arString2[1] := TO_STRING(iMedidor);
			arString2[2] := ' AND timestamps BETWEEN ';
			arString2[3] := CONCAT(CONCAT('("',RIGHT(STR:= DT_TO_STRING(Timestamp - T#3H), SIZE:= 19)),'"- INTERVAL 15 MINUTE)');
			arString2[4] := ' AND ';
			arString2[5] := CONCAT(CONCAT('("',RIGHT(STR:= DT_TO_STRING(Timestamp - T#3H), SIZE:= 19)), '");');
			
			sCmdEscreve1 := F_ConcatArray(sArray:= arString2);

			//Cria o array dos minutos e limpa o array atual
			FOR i := 1 TO 15 DO
				minute	:= DT_TO_SYSTEMTIME(Timestamp);
				MinutosAtuais[i] := WORD_TO_INT(minute.wMinute)-i+1;
				IF MinutosAtuais[i] < 0 THEN
					MinutosAtuais[i] := 60 + MinutosAtuais[i];
				END_IF
			END_FOR
			
			// call functionblock
			IF fbPLCDBCmd1.ExecuteDataReturn
				(
					hDBID := 1,
						pExpression := ADR(sCmdEscreve1),
						cbExpression := SIZEOF(sCmdEscreve1),
						pData := ADR(TagAProcurar),
						cbData := SIZEOF(TagAProcurar),
						pParameter := ADR(stPara),
						cbParameter := SIZEOF(stPara),
						nStartIndex := 0,
						nRecordCount := DINT_TO_UDINT(diCima),
						pReturnData := ADR(EstruturaBancoMinuto),
						cbReturnData := SIZEOF(EstruturaBancoMinuto),
						pRecords := ADR(nRecords))
			THEN
				IF fbPLCDBCmd1.bError THEN
					sMensagemErro2 := 'Nao conseguiu a tag';
				ELSE
					sMensagemErro2	:= 'Conseguiu a tag';
	
					
					FOR j := TO_INT(diBaixo) TO TO_INT(diCima) DO
						FOR i := 1 TO 15 DO
							minute	:= DT_TO_SYSTEMTIME(EstruturaBancoMinuto[j].Timestamp);
							IF (WORD_TO_INT(minute.wMinute) = MinutosAtuais[i] AND EstruturaBancoMinuto[j].Timestamp <> DT#1970-1-1-0:0:0) THEN
								Minutos[j].Medidor				:= EstruturaBancoMinuto[i].Medidor;
								Minutos[j].rConsumo1min			:= EstruturaBancoMinuto[i].rConsumo1min;
								Minutos[j].rDemanda1min 		:= EstruturaBancoMinuto[i].rDemanda1min;
								Minutos[j].rFatorDePotencia1min := EstruturaBancoMinuto[i].rFatorDePotencia1min;
								Minutos[j].Timestamp 			:= EstruturaBancoMinuto[i].Timestamp;
							END_IF
						END_FOR
						
						

					END_FOR
					
					iEstadoLeitura			:= 4;
				END_IF
			END_IF
		END_IF
		
		
		IF xDiaSelecionado THEN
			//Le os 15 minutos
			stPara.eParaType	:= E_ExpParameterType.Float32;
			stPara.nParaSize	:= SIZEOF(TagAProcurar);
			stPara.sParaName	:= 'rMedia15min';
			
				//RECUPERANDO DADOS DOS 15 MIN
			diBaixo	:= LOWER_BOUND(Media15Min, 1);
			diCima	:= UPPER_BOUND(Media15Min, 1);
	
			
			arString2[0] := 'SELECT * FROM dbexcelsior.media15min WHERE medidor=';
			arString2[1] := TO_STRING(iMedidor);
			arString2[2] := ' AND timestamps BETWEEN ';
			arString2[3] := CONCAT(CONCAT('("',LEFT(STR:=RIGHT(STR:= DT_TO_STRING(Timestamp - T#3H), SIZE:= 19) , SIZE:= 10)),'-00:00:00")');
			arString2[4] := ' AND ';
			arString2[5] := CONCAT(CONCAT('("',	RIGHT(STR:= DT_TO_STRING(Timestamp - T#3H), SIZE:= 19)), '");');
			
			sCmdEscreve2 := F_ConcatArray(sArray:= arString2);
			
			// call functionblock
			IF fbPLCDBCmd2.ExecuteDataReturn
				(
					hDBID := 1,
						pExpression := ADR(sCmdEscreve2),
						cbExpression := SIZEOF(sCmdEscreve2),
						pData := ADR(TagAProcurar),
						cbData := SIZEOF(TagAProcurar),
						pParameter := ADR(stPara),
						cbParameter := SIZEOF(stPara),
						nStartIndex := 0,
						nRecordCount := DINT_TO_UDINT(diCima),
						pReturnData := ADR(EstruturaBancoMedia15min),
						cbReturnData := SIZEOF(EstruturaBancoMedia15min),
						pRecords := ADR(nRecords))
			THEN
				IF fbPLCDBCmd2.bError THEN
					sMensagemErro2 := 'Nao conseguiu a tag';
				ELSE
					sMensagemErro2	:= 'Conseguiu a tag';
					iEstadoLeitura			:= 4;
	
					
					FOR j := TO_INT(diBaixo) TO TO_INT(diCima) DO
						IF EstruturaBancoMedia15min[j].Timestamp <> DT#1970-1-1-0:0:0 THEN
							times := DT_TO_SYSTEMTIME(EstruturaBancoMedia15min[j].Timestamp);
							posicao := PosicaoAtualdos15[times.wHour,times.wMinute];
							Media15Min[posicao].rMedia15min				:= EstruturaBancoMedia15min[j].rMedia15min;
							Media15Min[posicao].rFatorDePotencia15min	:= EstruturaBancoMedia15min[j].rFatorDePotencia15min;
							Media15Min[posicao].rConsumo15min			:= EstruturaBancoMedia15min[j].rConsumo15min;
							Media15Min[posicao].Timestamp				:= EstruturaBancoMedia15min[j].Timestamp;
							Media15Min[posicao].Medidor					:= EstruturaBancoMedia15min[j].Medidor;
						END_IF
					END_FOR
				END_IF
			END_IF
		END_IF
		
		IF xMesSelecionado THEN
			//Le os dias
			stPara.eParaType	:= E_ExpParameterType.Float32;
			stPara.nParaSize	:= SIZEOF(TagAProcurar);
			stPara.sParaName	:= 'rMediaDia';
			
			//RECUPERANDO DADOS DOS DIAS
			diBaixo	:= LOWER_BOUND(MediaDia, 1);
			diCima	:= UPPER_BOUND(MediaDia, 1);
	
			
			arString2[0] := 'SELECT * FROM dbexcelsior.mediadia WHERE medidor=';
			arString2[1] := TO_STRING(iMedidor);
			arString2[2] := ' AND timestamps BETWEEN ';
			arString2[3] := CONCAT(CONCAT('("',	LEFT(STR:= RIGHT(STR:= DT_TO_STRING(Timestamp - T#3H), SIZE:= 19), SIZE:= 7)),'-01-00:00:00")');
			arString2[4] := ' AND ';
			arString2[5] := CONCAT(CONCAT('("',	LEFT(STR:= RIGHT(STR:= DT_TO_STRING(Timestamp - T#3H), SIZE:= 19), SIZE:= 7)),'-01-23:59:59" + INTERVAL 1 MONTH - INTERVAL 1 DAY);');
			
			sCmdEscreve3 := F_ConcatArray(sArray:= arString2);
			
			// call functionblock
			IF fbPLCDBCmd3.ExecuteDataReturn
				(
					hDBID := 1,
						pExpression := ADR(sCmdEscreve3),
						cbExpression := SIZEOF(sCmdEscreve3),
						pData := ADR(TagAProcurar),
						cbData := SIZEOF(TagAProcurar),
						pParameter := ADR(stPara),
						cbParameter := SIZEOF(stPara),
						nStartIndex := 0,
						nRecordCount := DINT_TO_UDINT(diCima),
						pReturnData := ADR(EstruturaBancoMediaDia),
						cbReturnData := SIZEOF(EstruturaBancoMediaDia),
						pRecords := ADR(nRecords))
			THEN
				IF fbPLCDBCmd3.bError THEN
					sMensagemErro2 := 'Nao conseguiu a tag';
				ELSE
					sMensagemErro2	:= 'Conseguiu a tag';
					iEstadoLeitura			:= 4;
	
					
					FOR j := TO_INT(diBaixo) TO TO_INT(diCima) DO
							times := DT_TO_SYSTEMTIME(EstruturaBancoMediaDia[j].Timestamp);
							
							IF (EstruturaBancoMediaDia[j].Timestamp <> DT#1970-1-1-00:00:00) THEN
								MediaDia[times.wDay].rMediaDia				:= EstruturaBancoMediaDia[j].rMediaDia;
								MediaDia[times.wDay].rFatorDePotenciaDia	:= EstruturaBancoMediaDia[j].rFatorDePotenciaDia;
								MediaDia[times.wDay].rConsumoDia			:= EstruturaBancoMediaDia[j].rConsumoDia;
								MediaDia[times.wDay].Timestamp				:= EstruturaBancoMediaDia[j].Timestamp;
								MediaDia[times.wDay].Medidor				:= EstruturaBancoMediaDia[j].Medidor;
							END_IF
					END_FOR
				END_IF
			END_IF
		END_IF
		
		IF xAnoSelecionado THEN
			//Le os meses
			stPara.eParaType	:= E_ExpParameterType.Float32;
			stPara.nParaSize	:= SIZEOF(TagAProcurar);
			stPara.sParaName	:= 'rMediaMes';
			
			//RECUPERANDO DADOS DOS MESES
			diBaixo	:= LOWER_BOUND(MediaMes, 1);
			diCima	:= UPPER_BOUND(MediaMes, 1);
	
			
			arString2[0] := 'SELECT * FROM dbexcelsior.mediames WHERE medidor=';
			arString2[1] := TO_STRING(iMedidor);
			arString2[2] := ' AND timestamps BETWEEN ';
			arString2[3] := CONCAT(CONCAT('("',	LEFT(STR:= RIGHT(STR:= DT_TO_STRING(Timestamp - T#3H), SIZE:= 19), SIZE:= 4)),'-01-01-00:00:00")');
			arString2[4] := ' AND ';
			arString2[5] := CONCAT(CONCAT('("',	LEFT(STR:= RIGHT(STR:= DT_TO_STRING(Timestamp - T#3H), SIZE:= 19), SIZE:= 4)),'-12-31-23:59:59");');
			
			sCmdEscreve4 := F_ConcatArray(sArray:= arString2);
			
			// call functionblock
			IF fbPLCDBCmd4.ExecuteDataReturn
				(
					hDBID := 1,
						pExpression := ADR(sCmdEscreve4),
						cbExpression := SIZEOF(sCmdEscreve4),
						pData := ADR(TagAProcurar),
						cbData := SIZEOF(TagAProcurar),
						pParameter := ADR(stPara),
						cbParameter := SIZEOF(stPara),
						nStartIndex := 0,
						nRecordCount := DINT_TO_UDINT(diCima),
						pReturnData := ADR(EstruturaBancoMediaMes),
						cbReturnData := SIZEOF(EstruturaBancoMediaMes),
						pRecords := ADR(nRecords))
			THEN
				IF fbPLCDBCmd4.bError THEN
					sMensagemErro2 := 'Nao conseguiu a tag';
				ELSE
					sMensagemErro2	:= 'Conseguiu a tag';
					iEstadoLeitura			:= 4;
	
					
					FOR j := TO_INT(diBaixo) TO TO_INT(diCima) DO
						IF (EstruturaBancoMediaMes[j].Timestamp <> DT#1970-1-1-00:00:00) THEN
							times := DT_TO_SYSTEMTIME(EstruturaBancoMediaMes[j].Timestamp);
							MediaMes[times.wMonth].rMediaMes			:= EstruturaBancoMediaMes[j].rMediaMes;
							MediaMes[times.wMonth].rFatorDePotenciaMes	:= EstruturaBancoMediaMes[j].rFatorDePotenciaMes;
							MediaMes[times.wMonth].rConsumoMes			:= EstruturaBancoMediaMes[j].rConsumoMes;
							MediaMes[times.wMonth].Timestamp			:= EstruturaBancoMediaMes[j].Timestamp;
							MediaMes[times.wMonth].Medidor				:= EstruturaBancoMediaMes[j].Medidor;
						END_IF
					END_FOR
				END_IF
			END_IF
		END_IF
		
	4: // FechaConexao conexao
		IF fbSQLDatabase2.Disconnect() THEN

			xAtualizaInterno	:= FALSE;
			xAtualiza			:= FALSE;
			xTerminouLeitura	:= TRUE;
			
			IF fbSQLDatabase2.bError THEN
				iEstadoLeitura := 1;
			ELSE
				iEstadoLeitura := 1;
			END_IF
		END_IF
END_CASE
END_ACTION

END_FUNCTION_BLOCK

// FBs/MedicaoEnergia/FB_LeBancoDeDadosParaCSV
//{attribute 'hide_all_locals'}
FUNCTION_BLOCK FB_LeBancoDeDadosParaCSV
VAR_IN_OUT
	CSV15Min		: ARRAY[*] OF stMedia15min;
	CSVDia			: ARRAY[*] OF stMediaDia;
	CSVMes			: ARRAY[*] OF stMediaMes;
	CSVAno			: ARRAY[*] OF stMediaAno;
	CSVCorrente		: ARRAY[*] OF stCorrenteCSV;
END_VAR
VAR_INPUT
	xCriaTabelas		: BOOL;				// tenta criar a tabela
	iNumeroDataBase		: INT	:= 1;		// id do database
	xLeCSV15min			: BOOL;
	xLeCSVDia			: BOOL;
	xLeCSVMes			: BOOL;
	xLeCSVAno			: BOOL;
	xLeCSVCorrente		: BOOL;
END_VAR
VAR_OUTPUT
	xOcupado			: BOOL;
	xTodasTabelasCriadas: BOOL;
	xTerminei15min		: BOOL;
	xTermineiDia		: BOOL;
	xTermineiMes		: BOOL;
	xTermineiAno		: BOOL;
	xTermineiCorrente	: BOOL;
END_VAR
VAR
	//Cria table
	rtCria				: R_TRIG;
	xComecaCriarTabelas	: BOOL;
	xTabela1Criada		: BOOL;
	xTabela2Criada		: BOOL;
	xTabela3Criada		: BOOL;
	xTabela4Criada		: BOOL;
	xTabela5Criada		: BOOL;
	
	fbPLCDBCreate1	: FB_PLCDBCreateEvt(sNetID := '', tTimeout := T#30S);
	fbPLCDBCreate2	: FB_PLCDBCreateEvt(sNetID := '', tTimeout := T#30S);
	fbPLCDBCreate3	: FB_PLCDBCreateEvt(sNetID := '', tTimeout := T#30S);
	fbPLCDBCreate4	: FB_PLCDBCreateEvt(sNetID := '', tTimeout := T#30S);
	fbPLCDBCreate5	: FB_PLCDBCreateEvt(sNetID := '', tTimeout := T#30S);
	
	
	ColumnInfo1 : ARRAY[0..4] OF ST_ColumnInfo := [	(sName := 'rDemanda1min',	eType := E_ColumnType.REAL_,	nLength := 4),
													(sName := 'rFatorDePotencia1min',	eType := E_ColumnType.REAL_,	nLength := 4),
													(sName := 'rConsumo1min',	eType := E_ColumnType.REAL_,	nLength := 4),
													(sName := 'medidor',	eType := E_ColumnType.Integer, 	nLength := 2),
													(sName := 'timestamps', 	eType := E_ColumnType.DateTime, nLength := 4, sProperty := 'DEFAULT CURRENT_TIMESTAMP ON UPDATE CURRENT_TIMESTAMP')];
													
	ColumnInfo2 : ARRAY[0..4] OF ST_ColumnInfo := [	(sName := 'rMedia15min',eType := E_ColumnType.REAL_,	nLength := 4),
													(sName := 'rFatorDePotencia15min',	eType := E_ColumnType.REAL_,	nLength := 4),
													(sName := 'rConsumo15min',	eType := E_ColumnType.REAL_,	nLength := 4),
													(sName := 'medidor',	eType := E_ColumnType.Integer, 	nLength := 2),
													(sName := 'timestamps', 	eType := E_ColumnType.DateTime, nLength := 4, sProperty := 'DEFAULT CURRENT_TIMESTAMP ON UPDATE CURRENT_TIMESTAMP')];
													
	ColumnInfo3 : ARRAY[0..4] OF ST_ColumnInfo := [	(sName := 'rMediaDia',	eType := E_ColumnType.REAL_,	nLength := 4),
													(sName := 'rFatorDePotenciaDia',	eType := E_ColumnType.REAL_,	nLength := 4),
													(sName := 'rConsumoDia',	eType := E_ColumnType.REAL_,	nLength := 4),
													(sName := 'medidor',	eType := E_ColumnType.Integer, 	nLength := 2),
													(sName := 'timestamps', 	eType := E_ColumnType.DateTime, nLength := 4, sProperty := 'DEFAULT CURRENT_TIMESTAMP ON UPDATE CURRENT_TIMESTAMP')];
													
													
	ColumnInfo4 : ARRAY[0..4] OF ST_ColumnInfo := [	(sName := 'rMediaMes',	eType := E_ColumnType.REAL_,	nLength := 4),
													(sName := 'rFatorDePotenciaMes',	eType := E_ColumnType.REAL_,	nLength := 4),
													(sName := 'rConsumoMes',	eType := E_ColumnType.REAL_,	nLength := 4),
													(sName := 'medidor',	eType := E_ColumnType.Integer, 	nLength := 2),
													(sName := 'timestamps', 	eType := E_ColumnType.DateTime, nLength := 4, sProperty := 'DEFAULT CURRENT_TIMESTAMP ON UPDATE CURRENT_TIMESTAMP')];

	ColumnInfo5 : ARRAY[0..4] OF ST_ColumnInfo := [	(sName := 'rMediaAno',	eType := E_ColumnType.REAL_,	nLength := 4),
													(sName := 'rFatorDePotenciaAno',	eType := E_ColumnType.REAL_,	nLength := 4),
													(sName := 'rConsumoAno',	eType := E_ColumnType.REAL_,	nLength := 4),
													(sName := 'medidor',	eType := E_ColumnType.Integer, 	nLength := 2),
													(sName := 'timestamps', 	eType := E_ColumnType.DateTime, nLength := 4, sProperty := 'DEFAULT CURRENT_TIMESTAMP ON UPDATE CURRENT_TIMESTAMP')];
													
	//Le Valores
	sCmdEscreve					: STRING(1000);
	sMensagemErro				: STRING;
	EstruturaBancoMedia15min	: ARRAY[1..100000] OF stMedia15min;
	EstruturaBancoMediaDia		: ARRAY[1..2000] OF stMediaDia;
	EstruturaBancoMediaMes		: ARRAY[1..4000] OF stMediaMes;
	EstruturaBancoMediaAno		: ARRAY[1..700] OF stMediaAno;
	EstruturaBancoCorrente		: ARRAY[1..100000] OF stCorrenteCSV;
	nRecords					: UDINT;
	TagAProcurar				: REAL;
	diCima						: DINT;
	diBaixo						: DINT;
	iEstadoLeitura				: INT := 1;
	j							: UDINT;
	stPara						: ST_ExpParameter;
	fbSQLDatabase				: FB_SQLDatabaseEvt(sNetID := '', tTimeout := T#30S);
	fbPLCDBCmd1					: FB_PLCDBCmdEvt(sNetID := '', tTimeout := T#30S);
	fbPLCDBCmd2					: FB_PLCDBCmdEvt(sNetID := '', tTimeout := T#30S);
	fbPLCDBCmd3					: FB_PLCDBCmdEvt(sNetID := '', tTimeout := T#30S);
	fbPLCDBCmd4					: FB_PLCDBCmdEvt(sNetID := '', tTimeout := T#30S);
	fbPLCDBCmd5					: FB_PLCDBCmdEvt(sNetID := '', tTimeout := T#30S);
	rtLeitura1					: R_TRIG;
	rtLeitura2					: R_TRIG;
	rtLeitura3					: R_TRIG;
	rtLeitura4					: R_TRIG;
	rtLeitura5					: R_TRIG;
	xTemMais					: BOOL;
	xAtualizaInterno			: BOOL;	
	xLeCSV15minInterno			: BOOL;
	xLeCSVDiaInterno			: BOOL;
	xLeCSVMesInterno			: BOOL;
	xLeCSVAnoInterno			: BOOL;
	xLeCSVCorrenteInterno		: BOOL;									
													
END_VAR

//Criado Por Augusto Cazzanelli para o Projeto Excelsior
//GeraTabela();
IF xLicensaValida651641iih THEN
	rtLeitura1(CLK:= xLeCSV15min, Q=> );
	rtLeitura2(CLK:= xLeCSVDia, Q=> );
	rtLeitura3(CLK:= xLeCSVMes, Q=> );
	rtLeitura4(CLK:= xLeCSVAno, Q=> );
	rtLeitura5(CLK:= xLeCSVCorrente, Q=> );
	
	IF rtLeitura1.Q THEN
		xLeCSV15minInterno := TRUE;
		xTerminei15min := FALSE;
	END_IF
	
	IF rtLeitura2.Q THEN
		xLeCSVDiaInterno := TRUE;
		xTermineiDia := FALSE;
	END_IF
	
	IF rtLeitura3.Q THEN
		xLeCSVMesInterno := TRUE;
		xTermineiMes := FALSE;
	END_IF
	
	IF rtLeitura4.Q THEN
		xLeCSVAnoInterno := TRUE;
		xTermineiAno := FALSE;
	END_IF
	
	IF rtLeitura5.Q THEN
		xLeCSVCorrenteInterno := TRUE;
		xTermineiCorrente := FALSE;
	END_IF
	
	
	IF (xLeCSV15minInterno OR xLeCSVDiaInterno OR xLeCSVMesInterno OR xLeCSVAnoInterno OR xLeCSVCorrenteInterno) THEN
		xAtualizaInterno := TRUE;
	ELSE
		xAtualizaInterno := FALSE;
	END_IF
	
	LeValores();
END_IF;

ACTION GeraTabela:
(*
rtCria(CLK := xCriaTabelas, Q =>);

IF rtCria.q THEN
	xComecaCriarTabelas		:= TRUE;
	xOcupado				:= TRUE;
END_IF

IF xComecaCriarTabelas THEN
		//Cria a tabela com os minutos inidividuais de cada um dos 15 min
		IF fbPLCDBCreate1.Table
			(
				hDBID := INT_TO_UDINT(iNumeroDataBase),
					sTableName := 'minutos',
					pTableCfg := ADR(ColumnInfo1),
					cbTableCfg := SIZEOF(ColumnInfo1))
		THEN
			IF NOT fbPLCDBCreate1.bError  OR (fbPLCDBCreate1.bError AND fbPLCDBCreate1.ipTcResult.nEventId = 60) THEN
				xTabela1Criada := TRUE;
			ELSE
				xTabela1Criada := FALSE;
			END_IF
		END_IF


		//Cria a tabela com a media dos 15 min
		IF fbPLCDBCreate2.Table
		(
				hDBID := INT_TO_UDINT(iNumeroDataBase),
					sTableName := 'media15min',
					pTableCfg := ADR(ColumnInfo2),
					cbTableCfg := SIZEOF(ColumnInfo2))
		THEN
			IF NOT fbPLCDBCreate2.bError  OR (fbPLCDBCreate1.bError AND fbPLCDBCreate2.ipTcResult.nEventId = 60) THEN
				xTabela2Criada := TRUE;
			ELSE
				xTabela2Criada := FALSE;
			END_IF
		END_IF

		//Cria a tabela com a media dos dias
		IF fbPLCDBCreate3.Table
		(
				hDBID := INT_TO_UDINT(iNumeroDataBase),
					sTableName := 'mediadia',
					pTableCfg := ADR(ColumnInfo3),
					cbTableCfg := SIZEOF(ColumnInfo3))
		THEN
			IF NOT fbPLCDBCreate3.bError  OR (fbPLCDBCreate1.bError AND fbPLCDBCreate3.ipTcResult.nEventId = 60) THEN
				xTabela3Criada := TRUE;
			ELSE
				xTabela3Criada := FALSE;
			END_IF
		END_IF	

		//Cria a tabela com a media dos dias para a semana
		IF fbPLCDBCreate4.Table
		(
				hDBID := INT_TO_UDINT(iNumeroDataBase),
					sTableName := 'mediames',
					pTableCfg := ADR(ColumnInfo4),
					cbTableCfg := SIZEOF(ColumnInfo4))
		THEN
			IF NOT fbPLCDBCreate4.bError  OR (fbPLCDBCreate1.bError AND fbPLCDBCreate4.ipTcResult.nEventId = 60) THEN
				xTabela4Criada := TRUE;
			ELSE
				xTabela4Criada := FALSE;
			END_IF
		END_IF
		
		//Cria a tabela com a media do ano
		IF fbPLCDBCreate5.Table
		(
				hDBID := INT_TO_UDINT(iNumeroDataBase),
					sTableName := 'mediaano',
					pTableCfg := ADR(ColumnInfo5),
					cbTableCfg := SIZEOF(ColumnInfo5))
		THEN
			IF NOT fbPLCDBCreate5.bError  OR (fbPLCDBCreate5.bError AND fbPLCDBCreate5.ipTcResult.nEventId = 60) THEN
				xTabela5Criada := TRUE;
			ELSE
				xTabela5Criada := FALSE;
			END_IF
		END_IF



	
	IF (xTabela1Criada AND xTabela2Criada AND xTabela3Criada AND xTabela4Criada AND xTabela4Criada AND xTabela5Criada) THEN
		xComecaCriarTabelas		:= FALSE;
		xCriaTabelas	:= FALSE;
		xTodasTabelasCriadas := TRUE;
		xOcupado := FALSE;
	ELSE
		xCriaTabelas	:= FALSE;
		xComecaCriarTabelas		:= FALSE;
		xTodasTabelasCriadas := FALSE;
		xOcupado := FALSE;
	END_IF 
	
ELSE
	xOcupado := FALSE;
END_IF
*)
END_ACTION

ACTION LeValores:
CASE iEstadoLeitura OF
	1: //Esperando
		IF xAtualizaInterno THEN
			iEstadoLeitura := 3;
		END_IF

	2: //abre conexao
		IF fbSQLDatabase.Connect(INT_TO_UDINT(iNumeroDataBase)) THEN
			IF fbSQLDatabase.bError THEN
				IF fbSQLDatabase.ipTcResult.ipSourceInfo.sName = 'ADSERR_DEVICE_LICENSENOTFOUND' THEN
					// se der isso ele nao fica tentando e gerando uma caralhada de erro pq nao tem a lisença
					iEstadoLeitura := 0;
				ELSE
					iEstadoLeitura := 2;
				END_IF
			ELSE
				IF fbSQLDatabase.bConnected THEN
					iEstadoLeitura := 3;
				END_IF
			END_IF
		END_IF

	3: // Le os dados par ao CSV
		IF xLeCSV15minInterno THEN
			
			stPara.eParaType	:= E_ExpParameterType.Float32;
			stPara.nParaSize	:= SIZEOF(TagAProcurar);
			stPara.sParaName	:= 'rMedia15min';
		
			diBaixo	:= LOWER_BOUND(CSV15Min, 1);
			diCima	:= UPPER_BOUND(CSV15Min, 1);
			
			sCmdEscreve := 'SELECT * FROM dbexcelsior.media15min WHERE timestamps BETWEEN CURRENT_TIMESTAMP() - INTERVAL 14 DAY AND CURRENT_TIMESTAMP();';
			
			// call functionblock
			IF fbPLCDBCmd1.ExecuteDataReturn
				(
					hDBID := 1,
						pExpression := ADR(sCmdEscreve),
						cbExpression := SIZEOF(sCmdEscreve),
						pData := ADR(TagAProcurar),
						cbData := SIZEOF(TagAProcurar),
						pParameter := ADR(stPara),
						cbParameter := SIZEOF(stPara),
						nStartIndex := 0,
						nRecordCount := DINT_TO_UDINT(diCima),
						pReturnData := ADR(EstruturaBancoMedia15min),
						cbReturnData := SIZEOF(EstruturaBancoMedia15min),
						pRecords := ADR(nRecords))
			THEN
				IF fbPLCDBCmd1.bError THEN
					sMensagemErro := 'Nao conseguiu a tag';
				ELSE
					sMensagemErro	:= 'Conseguiu a tag';
					iEstadoLeitura			:= 4;
	
					
					FOR j := TO_UDINT(diBaixo) TO TO_UDINT(diCima) DO
						CSV15Min[j].rMedia15min					:= EstruturaBancoMedia15min[j].rMedia15min;
						CSV15Min[j].rFatorDePotencia15min		:= EstruturaBancoMedia15min[j].rFatorDePotencia15min;
						CSV15Min[j].rConsumo15min				:= EstruturaBancoMedia15min[j].rConsumo15min;
						CSV15Min[j].Timestamp					:= EstruturaBancoMedia15min[j].Timestamp;
						CSV15Min[j].Medidor						:= EstruturaBancoMedia15min[j].Medidor;
					END_FOR
					xTerminei15min := TRUE;
					xLeCSV15minInterno := FALSE;
				END_IF
			ELSE
				xTerminei15min := FALSE;
			END_IF
		END_IF
		
		IF xLeCSVDiaInterno THEN

			stPara.eParaType	:= E_ExpParameterType.Float32;
			stPara.nParaSize	:= SIZEOF(TagAProcurar);
			stPara.sParaName	:= 'rMediaDia';
		
			diBaixo	:= LOWER_BOUND(CSVDia, 1);
			diCima	:= UPPER_BOUND(CSVDia, 1);
			
			sCmdEscreve := 'SELECT * FROM dbexcelsior.mediadia WHERE timestamps BETWEEN CURRENT_TIMESTAMP() - INTERVAL 1 MONTH AND CURRENT_TIMESTAMP();';
			
			// call functionblock
			IF fbPLCDBCmd2.ExecuteDataReturn
				(
					hDBID := 1,
						pExpression := ADR(sCmdEscreve),
						cbExpression := SIZEOF(sCmdEscreve),
						pData := ADR(TagAProcurar),
						cbData := SIZEOF(TagAProcurar),
						pParameter := ADR(stPara),
						cbParameter := SIZEOF(stPara),
						nStartIndex := 0,
						nRecordCount := DINT_TO_UDINT(diCima),
						pReturnData := ADR(EstruturaBancoMediaDia),
						cbReturnData := SIZEOF(EstruturaBancoMediaDia),
						pRecords := ADR(nRecords))
			THEN
				IF fbPLCDBCmd2.bError THEN
					sMensagemErro := 'Nao conseguiu a tag';
				ELSE
					sMensagemErro	:= 'Conseguiu a tag';
					iEstadoLeitura			:= 4;
	
					
					FOR j := TO_UDINT(diBaixo) TO TO_UDINT(diCima) DO
						CSVDia[j].rMediaDia					:= EstruturaBancoMediaDia[j].rMediaDia;
						CSVDia[j].rFatorDePotenciaDia		:= EstruturaBancoMediaDia[j].rFatorDePotenciaDia;
						CSVDia[j].rConsumoDia				:= EstruturaBancoMediaDia[j].rConsumoDia;
						CSVDia[j].Timestamp					:= EstruturaBancoMediaDia[j].Timestamp;
						CSVDia[j].Medidor					:= EstruturaBancoMediaDia[j].Medidor;
					END_FOR
					xTermineiDia := TRUE;
					xLeCSVDiaInterno := FALSE;
				END_IF
			ELSE
				xTermineiDia := FALSE;
			END_IF
		END_IF
		
		IF xLeCSVMesInterno THEN
		
			stPara.eParaType	:= E_ExpParameterType.Float32;
			stPara.nParaSize	:= SIZEOF(TagAProcurar);
			stPara.sParaName	:= 'rMediaMes';
		
			diBaixo	:= LOWER_BOUND(CSVMes, 1);
			diCima	:= UPPER_BOUND(CSVMes, 1);
			
			sCmdEscreve := 'SELECT * FROM dbexcelsior.mediames WHERE timestamps BETWEEN CURRENT_TIMESTAMP() - INTERVAL 5 YEAR AND CURRENT_TIMESTAMP();';
			
			// call functionblock
			IF fbPLCDBCmd3.ExecuteDataReturn
				(
					hDBID := 1,
						pExpression := ADR(sCmdEscreve),
						cbExpression := SIZEOF(sCmdEscreve),
						pData := ADR(TagAProcurar),
						cbData := SIZEOF(TagAProcurar),
						pParameter := ADR(stPara),
						cbParameter := SIZEOF(stPara),
						nStartIndex := 0,
						nRecordCount := DINT_TO_UDINT(diCima),
						pReturnData := ADR(EstruturaBancoMediaMes),
						cbReturnData := SIZEOF(EstruturaBancoMediaMes),
						pRecords := ADR(nRecords))
			THEN
				IF fbPLCDBCmd3.bError THEN
					sMensagemErro := 'Nao conseguiu a tag';
				ELSE
					sMensagemErro	:= 'Conseguiu a tag';
					iEstadoLeitura			:= 4;
	
					
					FOR j := TO_UDINT(diBaixo) TO TO_UDINT(diCima) DO
						CSVMes[j].rMediaMes					:= EstruturaBancoMediaMes[j].rMediaMes;
						CSVMes[j].rFatorDePotenciaMes		:= EstruturaBancoMediaMes[j].rFatorDePotenciaMes;
						CSVMes[j].rConsumoMes				:= EstruturaBancoMediaMes[j].rConsumoMes;
						CSVMes[j].Timestamp					:= EstruturaBancoMediaMes[j].Timestamp;
						CSVMes[j].Medidor					:= EstruturaBancoMediaMes[j].Medidor;
					END_FOR
					xTermineiMes := TRUE;
					xLeCSVMesInterno := FALSE;
				END_IF
			ELSE
				xTermineiMes := FALSE;
			END_IF
		END_IF
		
		IF xLeCSVAnoInterno THEN
		
			stPara.eParaType	:= E_ExpParameterType.Float32;
			stPara.nParaSize	:= SIZEOF(TagAProcurar);
			stPara.sParaName	:= 'rMediaAno';
		
			diBaixo	:= LOWER_BOUND(CSVAno, 1);
			diCima	:= UPPER_BOUND(CSVAno, 1);
			
			sCmdEscreve := 'SELECT * FROM dbexcelsior.mediaano WHERE timestamps BETWEEN CURRENT_TIMESTAMP() - INTERVAL 10 YEAR AND CURRENT_TIMESTAMP();';
			
			// call functionblock
			IF fbPLCDBCmd4.ExecuteDataReturn
				(
					hDBID := 1,
						pExpression := ADR(sCmdEscreve),
						cbExpression := SIZEOF(sCmdEscreve),
						pData := ADR(TagAProcurar),
						cbData := SIZEOF(TagAProcurar),
						pParameter := ADR(stPara),
						cbParameter := SIZEOF(stPara),
						nStartIndex := 0,
						nRecordCount := DINT_TO_UDINT(diCima),
						pReturnData := ADR(EstruturaBancoMediaAno),
						cbReturnData := SIZEOF(EstruturaBancoMediaAno),
						pRecords := ADR(nRecords))
			THEN
				IF fbPLCDBCmd4.bError THEN
					sMensagemErro := 'Nao conseguiu a tag';
				ELSE
					sMensagemErro	:= 'Conseguiu a tag';
					iEstadoLeitura			:= 4;
	
					
					FOR j := TO_UDINT(diBaixo) TO TO_UDINT(diCima) DO
						CSVAno[j].rMediaAno					:= EstruturaBancoMediaAno[j].rMediaAno;
						CSVAno[j].rFatorDePotenciaAno		:= EstruturaBancoMediaAno[j].rFatorDePotenciaAno;
						CSVAno[j].rConsumoAno				:= EstruturaBancoMediaAno[j].rConsumoAno;
						CSVAno[j].Timestamp					:= EstruturaBancoMediaAno[j].Timestamp;
						CSVAno[j].Medidor					:= EstruturaBancoMediaAno[j].Medidor;
					END_FOR
					xTermineiAno := TRUE;
					xLeCSVAnoInterno := FALSE;
				END_IF
			ELSE
				xTermineiAno := FALSE;
			END_IF
		END_IF
		
		IF xLeCSVCorrenteInterno THEN
			
			stPara.eParaType	:= E_ExpParameterType.Float32;
			stPara.nParaSize	:= SIZEOF(TagAProcurar);
			stPara.sParaName	:= 'rCorrenteA';
		
			diBaixo	:= LOWER_BOUND(CSVCorrente, 1);
			diCima	:= UPPER_BOUND(CSVCorrente, 1);
			
			sCmdEscreve := 'SELECT * FROM dbexcelsior.corrente WHERE timestamps BETWEEN CURRENT_TIMESTAMP() - INTERVAL 14 DAY AND CURRENT_TIMESTAMP();';
			
			// call functionblock
			IF fbPLCDBCmd5.ExecuteDataReturn
				(
					hDBID := 1,
						pExpression := ADR(sCmdEscreve),
						cbExpression := SIZEOF(sCmdEscreve),
						pData := ADR(TagAProcurar),
						cbData := SIZEOF(TagAProcurar),
						pParameter := ADR(stPara),
						cbParameter := SIZEOF(stPara),
						nStartIndex := 0,
						nRecordCount := DINT_TO_UDINT(diCima),
						pReturnData := ADR(EstruturaBancoCorrente),
						cbReturnData := SIZEOF(EstruturaBancoCorrente),
						pRecords := ADR(nRecords))
			THEN
				IF fbPLCDBCmd5.bError THEN
					sMensagemErro := 'Nao conseguiu a tag';
				ELSE
					sMensagemErro	:= 'Conseguiu a tag';
					iEstadoLeitura			:= 1;
	
					
					FOR j := TO_UDINT(diBaixo) TO TO_UDINT(diCima) DO
						CSVCorrente[j].rCorrenteA				:= EstruturaBancoCorrente[j].rCorrenteA;
						CSVCorrente[j].rCorrenteB				:= EstruturaBancoCorrente[j].rCorrenteB;
						CSVCorrente[j].rCorrenteC				:= EstruturaBancoCorrente[j].rCorrenteC;
						CSVCorrente[j].rCorrenteMedia			:= EstruturaBancoCorrente[j].rCorrenteMedia;
						CSVCorrente[j].Timestamp				:= EstruturaBancoCorrente[j].Timestamp;
						CSVCorrente[j].Medidor					:= EstruturaBancoCorrente[j].Medidor;
					END_FOR
					xTermineiCorrente := TRUE;
					xLeCSVCorrenteInterno := FALSE;
				END_IF
			ELSE
				xTermineiCorrente := FALSE;
			END_IF
		END_IF

		
		IF NOT xLeCSV15minInterno AND NOT xLeCSVDiaInterno AND NOT xLeCSVMesInterno AND NOT xLeCSVAnoInterno AND NOT xLeCSVCorrenteInterno THEN
			iEstadoLeitura := 1;
		END_IF
		


	4: // FechaConexao conexao
		IF fbSQLDatabase.Disconnect() THEN
			
			
			IF fbSQLDatabase.bError THEN
				iEstadoLeitura := 1;
			ELSE
				iEstadoLeitura := 1;
			END_IF
		END_IF
END_CASE
END_ACTION

END_FUNCTION_BLOCK

// FBs/MedicaoEnergia/FB_NomesMedidoresPM2100
FUNCTION_BLOCK FB_NomesMedidoresPM2100
VAR_IN_OUT
	stPM2100	: ARRAY[*] OF st_PM2100_485_Schneider;
END_VAR
VAR_INPUT
	xInicia			: BOOL;
	xCriaTabela		: BOOL;
	iNumeroDataBase	: INT		:= 1;
	sNomeDataBase	: STRING	:= 'nomes';
END_VAR
VAR_OUTPUT
	xOcupado	: BOOL;
END_VAR
VAR
	//Cria table
	rtCria			: R_TRIG;
	xCria			: BOOL;
	fbPLCDBCreate	: FB_PLCDBCreateEvt(sNetID := '', tTimeout := T#30S);
	ColumnInfo : ARRAY[0..2] OF ST_ColumnInfo := [(sName := 'Medidor', eType := E_ColumnType.Integer, nLength := 8, sProperty := 'IDENTITY(1,1)'),
												  (sName := 'Tag', eType := E_ColumnType.NVarChar, nLength := 80, sProperty := 'DEFAULT $'SEMTAG$''),
												  (sName := 'Funcao', eType := E_ColumnType.NVarChar, nLength := 80, sProperty := 'DEFAULT $'NADA$'')];
												  

	//Le os nomes
	xFirstScan		: BOOL := TRUE;
	xLe				: BOOL;
	sCmd			: STRING(1000);
	sTag1			: STRING;
	TagAProcurar	: STRING(80);
	sMensagemErro1	: STRING;
	iIndexGrava		: INT := 0;
	iAux			: DINT;
	diCima			: DINT;
	diBaixo			: DINT;
	nRecords		: UDINT;
	Anterior		: ARRAY[0..999] OF st_PM2100_485_Schneider;
	stPara			: ST_ExpParameter;
	EstruturaBancoLe: ARRAY[0..999] OF stConfigNomeMedidorDB;
	eEstado			: enum_LeituradosNomes := enum_LeituradosNomes.eEsperando;
	fbSQLDatabase	: FB_SQLDatabaseEvt(sNetID := '', tTimeout := T#30S);
	fbPLCDBCmd		: FB_PLCDBCmdEvt(sNetID := '', tTimeout := T#30S);
	
	
	//Gera os Telerruptores
	diParteBaixa		: DINT;
	diParteAlta			: DINT;
	i					: INT;
	xGeraMedidores		: BOOL;
	xEscreve			: BOOL;
	xEscreveAux			: BOOL;
	rtEscrita			: R_TRIG;	
	EstruturaBanco		: ARRAY[0..999] OF stConfigNomeMedidorDB;
	fbPLCDBWrite		: FB_PLCDBWriteEvt(sNetID := '', tTimeout := T#30S); //Bloco para gravar no banco de dados
	ColumnNamesGrava	: ARRAY[0..2] OF STRING(50) := ['Medidor',
														'Tag',
														'Funcao'
														];
	//Grava Nomes Novos
	j				: INT;
	xGrava			: BOOL;
	xAberto			: BOOL;
	sCmd2			: STRING(1000);
	sMensagemErro2	: STRING;
	Nome			: STRING;
	Vazio			: STRING := '';
	Tag				: STRING;
	Funcao			: STRING;
	arrStr			: ARRAY[1..10] OF STRING(255);
	eEstadoGrava	: enum_GravaNomes := enum_GravaNomes.eEsperando;
	fbSqlCommand		: FB_SQLCommandEvt(sNetID := '', tTimeout := T#30S);
	fbSQLDatabase2	: FB_SQLDatabaseEvt(sNetID := '', tTimeout := T#30S);
	
END_VAR



IF xFirstScan THEN
	xLe := TRUE;
	xCriaTabela := TRUE;
END_IF

IF xInicia THEN
	xLe := TRUE;
	eEstado := enum_LeituradosNomes.eEsperando;
END_IF




GeraTabela();
//GeraOsMedidores();
LeNomes();
GravaValores();

xFirstScan := FALSE;

ACTION GeraOsMedidores:

diParteBaixa	:= LOWER_BOUND(stPM2100, 1);
diParteAlta		:= UPPER_BOUND(stPM2100, 1);

IF xGeraMedidores THEN

	xEscreve := TRUE;
	rtEscrita(CLK := xEscreve, Q =>);

	IF rtEscrita.q THEN
		xEscreveAux						:= TRUE;
		xOcupado						:= TRUE;
		i := DINT_TO_INT(diParteBaixa);
	END_IF

	IF xEscreveAux THEN
		EstruturaBanco[i].Tag := CONCAT('P', INT_TO_STRING(i+1));
		EstruturaBanco[i].Medidor := INT_TO_DINT(i);
		
		IF fbPLCDBWrite.WriteStruct
		(
			hDBID := INT_TO_UDINT(iNumeroDataBase),
				sTableName := sNomeDataBase,
				pRecord := ADR(EstruturaBanco[i]),
				cbRecord := SIZEOF(EstruturaBanco[i]),
				pColumnNames := ADR(ColumnNamesGrava),
				cbColumnNames := SIZEOF(ColumnNamesGrava))
		THEN
			i := i +1;
		ELSE
			IF fbPLCDBWrite.bError THEN
				IF fbPLCDBWrite.ipTcResult.nEventId = 61 THEN
					xCriaTabela := TRUE;
				END_IF
			END_IF
		END_IF
		
		IF i > diParteAlta THEN
			xOcupado	:= FALSE;
			xEscreve 	:= FALSE;
			rtEscrita(CLK := xEscreve, Q =>);
			xEscreveAux	:= FALSE;
			xGeraMedidores := FALSE;
			i := DINT_TO_INT(diParteBaixa);
			
			xLe := TRUE;
			eEstado := enum_LeituradosNomes.eEsperando;
		END_IF

	END_IF
END_IF
END_ACTION

ACTION GeraTabela:

rtCria(CLK := xCriaTabela, Q =>);

IF rtCria.q THEN
	xCria		:= TRUE;
	xOcupado	:= TRUE;
END_IF

IF xCria THEN

	IF fbPLCDBCreate.Table
		(
			hDBID := INT_TO_UDINT(iNumeroDataBase),
				sTableName := sNomeDataBase,
				pTableCfg := ADR(ColumnInfo),
				cbTableCfg := SIZEOF(ColumnInfo))
	THEN
		xCria		:= FALSE;
		xCriaTabela	:= FALSE;
		xOcupado	:= FALSE;
		xGeraMedidores	:= TRUE;
		i			:= 0;
	END_IF

END_IF
END_ACTION

ACTION GravaValores:
CASE eEstadoGrava OF
		enum_GravaNomes.eEsperando: //Esperando
			IF xGrava THEN
				IF xAberto THEN
					eEstadoGrava := enum_GravaNomes.eCriaComando;
				ELSE
					eEstadoGrava := enum_GravaNomes.eAbreConexao;
				END_IF
				
			END_IF
			
